FUNCTION "COOLANT" : VOID	// FC 50
TITLE = Coolant high pressure-KmDruckerhöhung
AUTHOR : A.Petz
VERSION : 0.6
VAR_INPUT
  iPnennV : INT ;	//Nenndruck des KmHochdruckventils bei 10V [Bar]
  iPMin : INT ;	//Min-Grenze für Anwahl Druckstufe [Bar]
  iPMax : INT ;	//Max-Grenze für Anwahl Druckstufe [Bar]
  iAfl : BYTE ;	//Meßwertauflösung (0:11+Vz,1:12+Vz,2:13+Vz,3-FF:15+Vz)
  iRmoDs : BOOL ;	//Rückmeldungen an LPlc ohne direkte KmDruckschalterabfrage
  iRmoFls : BOOL ;	//Rückmeldungen an LPlc ohne direkte KmDurchfluss-Schalterabfrage
  iFixedPressure : BOOL ;	//Anwahl für Druckerhöhungsstation mit fester Druckstufe IKZ (=TRUE)
END_VAR
VAR_TEMP
  iPlc : STRUCT 	//Signale von LeitPLC (aus DB111)
   machine_on : BOOL ;	//vonLPlc:Maschine bereit
   workroomdoor : BOOL ;	//vonLPlc:Arbeitsraumtüren geschlossen+verriegelt
   alarm_quit : BOOL ;	//vonLPlc:Störung, Alarm quittieren (Alarm Cancel)
   x : BOOL ;	//vonLPlc:
   coo_backflow : BOOL ;	//vonLPlc:Kühlmittelrückförderpumpe läuft
   pneumatic_pressure : BOOL ;	//vonLPlc:Pneumatik-(Luft-)druck vorhanden
   xa : BOOL ;	//vonLPlc:
   xb : BOOL ;	//vonLPlc:
   strobe_coo_pressure : BOOL ;	//vonLPlc:Strobe Druckumschaltung
   x_1 : BOOL ;	//vonLPlc:
   x_2 : BOOL ;	//vonLPlc:
   x_3 : BOOL ;	//vonLPlc:
   x_4 : BOOL ;	//vonLPlc:
   x_5 : BOOL ;	//vonLPlc:
   x_6 : BOOL ;	//vonLPlc:
   x_7 : BOOL ;	//vonLPlc:
   coolant1_m8 : BOOL ;	//vonLPlc:Anford. Kühmittel 1 (M8), Niederdruck
   coolant2_m7 : BOOL ;	//vonLPlc:Anford. Kühmittel 2 (M7), Hochdruck
   spraygun : BOOL ;	//vonLPlc:Anford. Spülpistole
   flush_lasercover : BOOL ;	//vonLPlc:Anford.Spülung Laservermessungsabdeckung
   flush_workpiece1 : BOOL ;	//vonLPlc:Anford.für Dach=Werkstückspülung
   flush_pallet_carrier : BOOL ;	//vonLPlc:Anford.Tischspülung bei PalWechsel
   flush_workroomdoor : BOOL ;	//vonLPlc:Anford.Arbeitsraumtür spülen
   flush_setupstation : BOOL ;	//vonLPlc:Anford.Rüstplatzspülung(Vorrichtung)
   x_16 : BOOL ;	//vonLPlc:
   x_17 : BOOL ;	//vonLPlc:
   x_18 : BOOL ;	//vonLPlc:
   x_19 : BOOL ;	//vonLPlc:
   x_20 : BOOL ;	//vonLPlc:
   x_21 : BOOL ;	//vonLPlc:
   x_22 : BOOL ;	//vonLPlc:
   x_23 : BOOL ;	//vonLPlc:
   PSoll : BYTE ;	//vonLPlc:Anwahl Druckstufe, BCD
   resBy : BYTE ;	//vonLPlc:Reserve Anwahl Druckstufe
  END_STRUCT ;
  oPlc : STRUCT 	//Signale an LeitPLC (DB112)
   ack_coolant1_m8 : BOOL ;	//anLPlc:Kühlmittel 1 (Niederdruck) ok
   ack_coolant2_m7 : BOOL ;	//anLPlc:Kühlmittel 2 (Hochdruck) ok
   message_flag : BOOL ;	//anLPlc:Warnung an Bediener, zB.Wasserstand
   no_emergency_stop : BOOL ;	//anLPlc:Fehler in Ksa, NotAus Masch.erforderlich
   no_spindle_feed_stop : BOOL ;	//anLPlc:Anford.SpiVs Halt durch Fehler in Ksa
   no_spindle_feed_stp_g0 : BOOL ;	//anLPlc:Anford.SpiVs Halt durch Fehler in Ksa bei nächst.G0
   no_diagnostic_alarm : BOOL ;	//anLPlc:Desina-Schalterüberwachung LOW-aktiv
   mode_auto : BOOL ;	//anLPlc:Kühlschmierstoffanlage in Betriebsart Automatik
   circuit_open_stop : BOOL ;	//anLPlc:Km Motorschutz gefallen, Masch.Halt
   circuit_open_msg : BOOL ;	//anLPlc:Km Motorschutz gefallen, Meldung
   x12 : BOOL ;	//anLPlc:Reserve Ksa max.Füllstand
   x13 : BOOL ;	//anLPlc:Reserve Ksa Warnung .min.Füllstand
   x14 : BOOL ;	//anLPlc:Reserve Ksa min.Füllstand, Masch.Halt
   x15 : BOOL ;	//anLPlc:Reserve Ksa Ende Papierbandfilter
   x16 : BOOL ;	//anLPlc:Reserve Ksa Warnung Ende Papierbandfilter
   x17 : BOOL ;	//anLPlc:Reserve
   PSoll : BYTE ;	//anLPlc:Rückmeldung Druckstufe, BCD
   resBy : BYTE ;	//anLPlc:Reserve Rückmeldung Druckstufe
  END_STRUCT ;
  s : STRUCT 	//statische da gerettete Lokaldaten
   PSoll : INT ;	//stat:letzter gespeicherter KmSolldruck
   PSollAlt : INT ;	//stat:letzter gespeich.KmSolldruck (alt, für Änderungserfassung)
   PSollAA : INT ;	//stat:letzter gespeich.KmSolldruck, berechnet für AA
   P20AA : INT ;	//stat:Solldruck 20Bar, berechnet für AA
   P40AA : INT ;	//stat:Solldruck 40Bar, berechnet für AA
   fk : ARRAY  [0 .. 15 ] OF //stat:Flankenhilfsmerker
   BOOL ;
   hvFEin : BOOL ;	//stat:KmHauptventil Fehler:Einschaltüberwachung
   hvFUnt : BOOL ;	//stat:KmHauptventil Fehler:Unterbrechungsüberwachung
   kmdFEin : BOOL ;	//stat:KmSystem=Niederdruck Fehler:Einschaltüberwachung
   kmdFUnt : BOOL ;	//stat:KmSystem=Niederdruck Fehler:Unterbrechungsüberwachung
   FlFEin : BOOL ;	//stat:KmDurchfluss Fehler:Einschaltüberwachung
   FlFUnt : BOOL ;	//stat:KmDurchfluss Fehler:Unterbrechungsüberwachung
   x_6 : BOOL ;	//stat:
   x_7 : BOOL ;	//stat:
   x_8 : BOOL ;	//stat:
   x_9 : BOOL ;	//stat:
   x_10 : BOOL ;	//stat:
   x_11 : BOOL ;	//stat:
   x_12 : BOOL ;	//stat:
   x_13 : BOOL ;	//stat:
   x_14 : BOOL ;	//stat:
   x_15 : BOOL ;	//stat:
  END_STRUCT ;
  svAR1 : DWORD ;	//Rettregister für AR1
  WertAA : INT ;	//Sollwert für Analogausgabe, ohne Meßwertauflösung
  LOp1 : BOOL ;	//lokaler Operationsmerker 1, Zwischenmerker
  LOp2 : BOOL ;	//lokaler Operationsmerker 2, Zwischenmerker
  LOp3 : BOOL ;	//lokaler Operationsmerker 3, Zwischenmerker
  fa : BOOL ;	//Freigabe Ausgänge
  no_coo_pressure : BOOL ;	//keine Km-Niederdruck Störung
  no_coo_flow : BOOL ;	//keine Km-Durchfluss Störung
  need_ventilate : BOOL ;	//Entlüftung wird benötigt
  ilp_ventilated : BOOL ;	//Anlage entlüftet
  shutdown_m7_opendoor : BOOL ;	//Abschaltung M7 über Öffnen der Arbeitsraumtüre
END_VAR
BEGIN
NETWORK
TITLE = Lokaldaten laden
      TAR1  #svAR1;
      LAR1  P##iPlc;
      L     DB111.DBD 0;
      T     LD [AR1,P#0.0];
      L     DB111.DBW 4;
      T     LW [AR1,P#4.0];
      LAR1  P##oPlc;
      L     DB112.DBW 0;
      T     LW [AR1,P#0.0];
      L     DB112.DBW 6;
      T     LW [AR1,P#2.0];
      LAR1  P##s;
      L     DB50.DBD 0;
      T     LD [AR1,P#0.0];
      L     DB50.DBD 4;
      T     LD [AR1,P#4.0];
      L     DB50.DBD 8;
      T     LD [AR1,P#8.0];
      L     DB50.DBW 12;
      T     LW [AR1,P#12.0];
      LAR1  #svAR1;
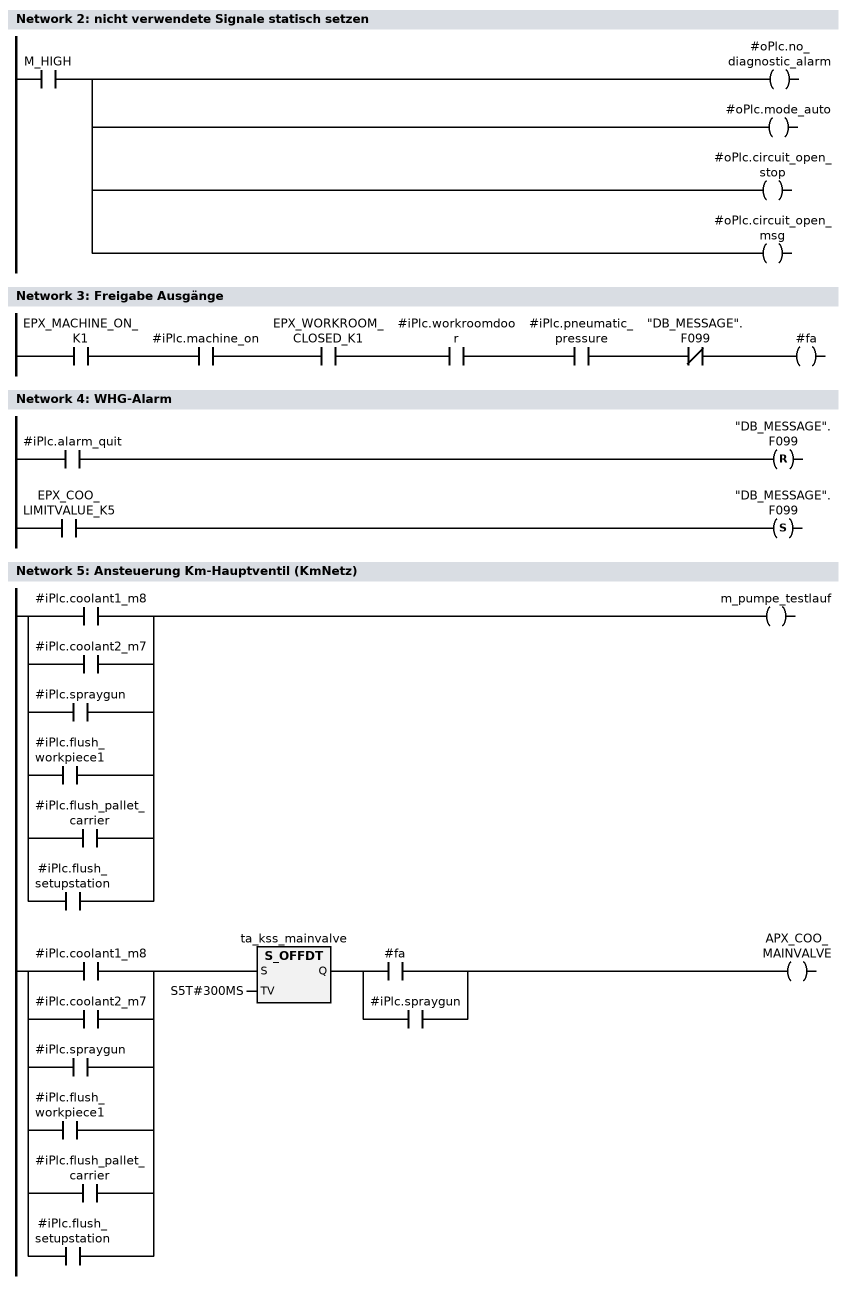
NETWORK
TITLE = nicht verwendete Signale statisch setzen 
      A     "M_HIGH";
      =     #oPlc.no_diagnostic_alarm;
      =     #oPlc.mode_auto;
      =     #oPlc.circuit_open_stop;
      =     #oPlc.circuit_open_msg;
NETWORK
TITLE = Freigabe Ausgänge
      A     "EPX_MACHINE_ON_K1";
      A     #iPlc.machine_on;
      A     "EPX_WORKROOM_CLOSED_K1";
      A     #iPlc.workroomdoor;
      A     #iPlc.pneumatic_pressure;
      AN    "DB_MESSAGE".F099;
      =     #fa;
NETWORK
TITLE = WHG-Alarm
      A     #iPlc.alarm_quit;
      R     "DB_MESSAGE".F099;
      A     "EPX_COO_LIMITVALUE_K5";
      S     "DB_MESSAGE".F099;
      NOP   0;
NETWORK
TITLE = Ansteuerung Km-Hauptventil (KmNetz)
//Bei Aktivierung der Sppritzpistole, wird nicht darauf geachtet ob die 
//Arbeitsraumtüren bzw. Rüstplatztüren geöffnet bzw. geschlossen sind, da dieses 
//PLC-seitig durchgeführt wird.
      O     #iPlc.coolant1_m8;
      O     #iPlc.coolant2_m7;
      O     #iPlc.spraygun;
      O     #iPlc.flush_workpiece1;
      O     #iPlc.flush_pallet_carrier;
      O     #iPlc.flush_setupstation;
      =     L 32.0;
      A(;
      A     L 32.0;
      L     S5T#300MS;
      SF    "ta_kss_mainvalve";
      NOP   0;
      NOP   0;
      NOP   0;
      A     "ta_kss_mainvalve";
      );
      A(;
      O     #fa;
      O     #iPlc.spraygun;
      );
      =     "APX_COO_MAINVALVE";
      A     L 32.0;
      BLD   102;
      =     "m_pumpe_testlauf";
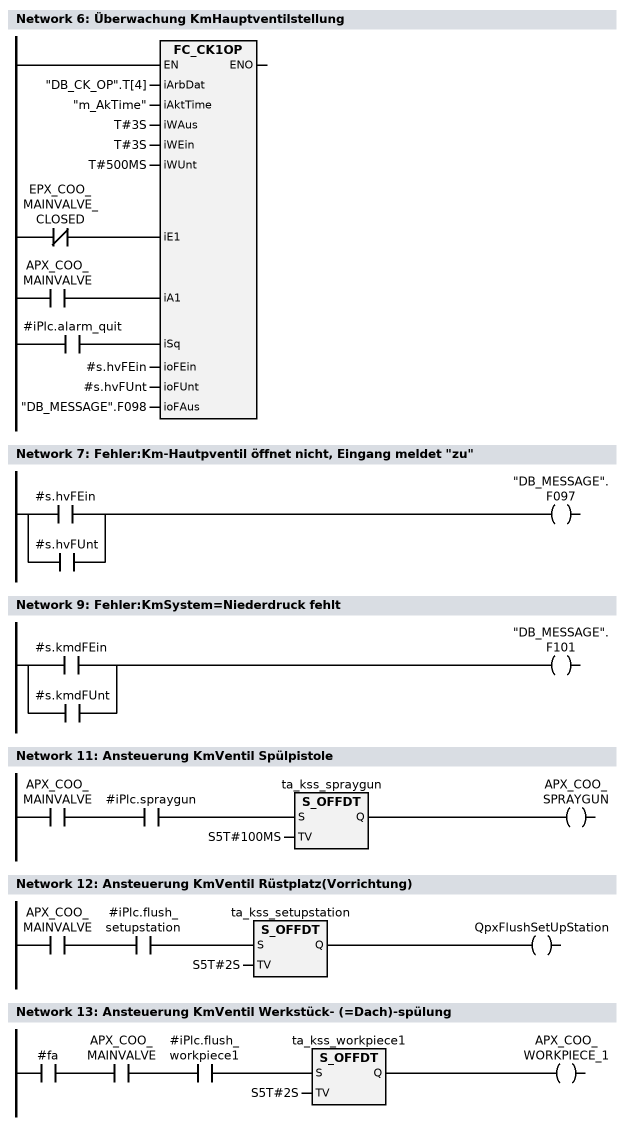
NETWORK
TITLE = Überwachung KmHauptventilstellung
//Koaxialventil
//Fabrikat: müller coax  Typ: 5-VMK32
//Das Ventil ist mit einem Endschalter ausgerüstet, welcher die 
//"geschlossen"-Position überwacht.
      AN    "EPX_COO_MAINVALVE_CLOSED";
      =     L 32.0;
      BLD   103;
      A     "APX_COO_MAINVALVE";
      =     L 32.1;
      BLD   103;
      A     #iPlc.alarm_quit;
      =     L 32.2;
      BLD   103;
      CALL  "FC_CK1OP" (
           iArbDat                  := "DB_CK_OP".T[4],
           iAktTime                 := "m_AkTime",
           iWAus                    := T#3S,
           iWEin                    := T#3S,
           iWUnt                    := T#500MS,
           iE1                      := L 32.0,
           iA1                      := L 32.1,
           iSq                      := L 32.2,
           ioFEin                   := #s.hvFEin,
           ioFUnt                   := #s.hvFUnt,
           ioFAus                   := "DB_MESSAGE".F098);
      NOP   0;
NETWORK
TITLE = Fehler:Km-Hautpventil öffnet nicht, Eingang meldet "zu"
//Koaxialventil
//Fabrikat: müller coax  Typ: 5-VMK32
//Das Ventil ist mit einem Endschalter ausgerüstet, welcher die 
//"geschlossen"-Position überwacht.
      O     #s.hvFEin;
      O     #s.hvFUnt;
      =     "DB_MESSAGE".F097;
NETWORK
TITLE = Überwachung KmSystem=Niederdruck
//Drucküberwachung wird zeitverzögert nach Entlüftung aktiviert, da die Anlage 
//Zeit zum Entlüften braucht.(Entlüftung nur bei geschlossener Arbeitsraumtüre)
      A     "EPX_COO_PRESSURE_P=MAX";
      A     "EPX_MACHINE_ON_K1";
      =     L 32.0;
      BLD   103;
      A     "APX_COO_MAINVALVE";
      =     L 32.1;
      BLD   103;
      A     #iPlc.alarm_quit;
      =     L 32.2;
      BLD   103;
      A(;
      A(;
      A     "ta_pressureless";
      L     S5T#1S;
      SD    "te_aktiv_monit_pressure";
      NOP   0;
      NOP   0;
      NOP   0;
      A     "te_aktiv_monit_pressure";
      );
      S     #ilp_ventilated;
      A     #need_ventilate;
      R     #ilp_ventilated;
      A     #ilp_ventilated;
      );
      JNB   _001;
      CALL  "FC_CK1OP" (
           iArbDat                  := "DB_CK_OP".T[5],
           iAktTime                 := "m_AkTime",
           iWAus                    := T#10S,
           iWEin                    := T#5S,
           iWUnt                    := T#2S,
           iE1                      := L 32.0,
           iA1                      := L 32.1,
           iSq                      := L 32.2,
           ioFEin                   := #s.kmdFEin,
           ioFUnt                   := #s.kmdFUnt,
           ioFAus                   := "DB_MESSAGE".F102);
_001: NOP   0;
NETWORK
TITLE = Fehler:KmSystem=Niederdruck fehlt
      O     #s.kmdFEin;
      O     #s.kmdFUnt;
      =     "DB_MESSAGE".F101;
NETWORK
TITLE = Aktivierung Kühlschmierstoffzufuhr_1 (externe - Spritzdüsen)
//Entlüftung der Anlage über M8 ist erst möglich wenn die Arbeitsraumtüre 
//geschlossen ist.
//Bei Abschaltung M7 über Türe öffnen wird ebenfalls ein Signal zur 
//erforderlichen 
//Entlüftung ausgegeben, da M7 Plc seitig nicht abfällt wenn Türe geöffnet wird.
      O(;
      A     #fa;
      A     "APX_COO_MAINVALVE";
      A     #iPlc.coolant1_m8;
      L     S5T#2S;
      SF    "ta_kss_km1";
      NOP   0;
      NOP   0;
      NOP   0;
      A     "ta_kss_km1";
      );
      O(;
      A(;
      A(;
      A(;
      A(;
      A     #iPlc.coolant2_m7;
      S     #shutdown_m7_opendoor;
      AN    #iPlc.workroomdoor;
      R     #shutdown_m7_opendoor;
      A     #shutdown_m7_opendoor;
      );
      FN    "m_fn_m7opendoor";
      O(;
      A(;
      O     #iPlc.coolant2_m7;
      O     #iPlc.flush_pallet_carrier;
      O     #iPlc.spraygun;
      );
      FN    "m_fn_m7S";
      );
      O(;
      A     "EPX_MACHINE_ON_K1";
      FP    "m_fp_masch_on";
      );
      );
      S     #need_ventilate;
      A     "ta_pressureless";
      R     #need_ventilate;
      A     #need_ventilate;
      );
      A     #iPlc.workroomdoor;
      L     S5T#2S;
      SF    "ta_pressureless";
      NOP   0;
      NOP   0;
      NOP   0;
      A     "ta_pressureless";
      );
      AN    "APX_COO_MAINVALVE";
      );
      =     "APX_COO_COOLANT1_(M8)";
NETWORK
TITLE = Ansteuerung KmVentil Spülpistole
      A     "APX_COO_MAINVALVE";
      A     #iPlc.spraygun;
      L     S5T#100MS;
      SF    "ta_kss_spraygun";
      NOP   0;
      NOP   0;
      NOP   0;
      A     "ta_kss_spraygun";
      =     "APX_COO_SPRAYGUN";
NETWORK
TITLE = Ansteuerung KmVentil Rüstplatz(Vorrichtung)
      A     "APX_COO_MAINVALVE";
      A     #iPlc.flush_setupstation;
      L     S5T#2S;
      SF    "ta_kss_setupstation";
      NOP   0;
      NOP   0;
      NOP   0;
      A     "ta_kss_setupstation";
      =     "QpxFlushSetUpStation";
NETWORK
TITLE = Ansteuerung KmVentil Werkstück- (=Dach)-spülung
      A     #fa;
      A     "APX_COO_MAINVALVE";
      A     #iPlc.flush_workpiece1;
      L     S5T#2S;
      SF    "ta_kss_workpiece1";
      NOP   0;
      NOP   0;
      NOP   0;
      A     "ta_kss_workpiece1";
      =     "APX_COO_WORKPIECE_1";
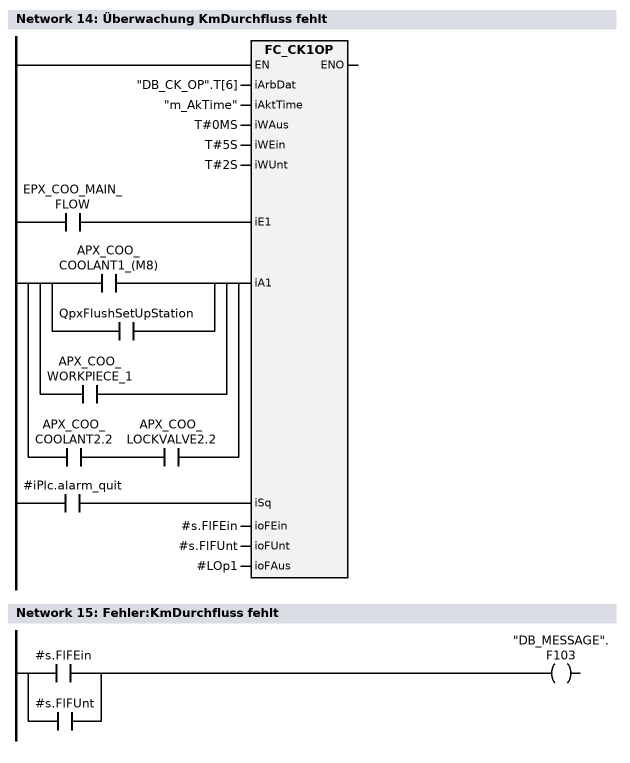
NETWORK
TITLE = Überwachung KmDurchfluss fehlt
      A     "EPX_COO_MAIN_FLOW";
      =     L 32.0;
      BLD   103;
      A(;
      O     "APX_COO_COOLANT1_(M8)";
      O     "QpxFlushSetUpStation";
      O     "APX_COO_WORKPIECE_1";
      O;
      A     "APX_COO_COOLANT2.2";
      A     "APX_COO_LOCKVALVE2.2";
      );
      =     L 32.1;
      BLD   103;
      A     #iPlc.alarm_quit;
      =     L 32.2;
      BLD   103;
      CALL  "FC_CK1OP" (
           iArbDat                  := "DB_CK_OP".T[6],
           iAktTime                 := "m_AkTime",
           iWAus                    := T#0MS,
           iWEin                    := T#5S,
           iWUnt                    := T#2S,
           iE1                      := L 32.0,
           iA1                      := L 32.1,
           iSq                      := L 32.2,
           ioFEin                   := #s.FlFEin,
           ioFUnt                   := #s.FlFUnt,
           ioFAus                   := #LOp1);
      NOP   0;
NETWORK
TITLE = Fehler:KmDurchfluss fehlt
      O     #s.FlFEin;
      O     #s.FlFUnt;
      =     "DB_MESSAGE".F103;
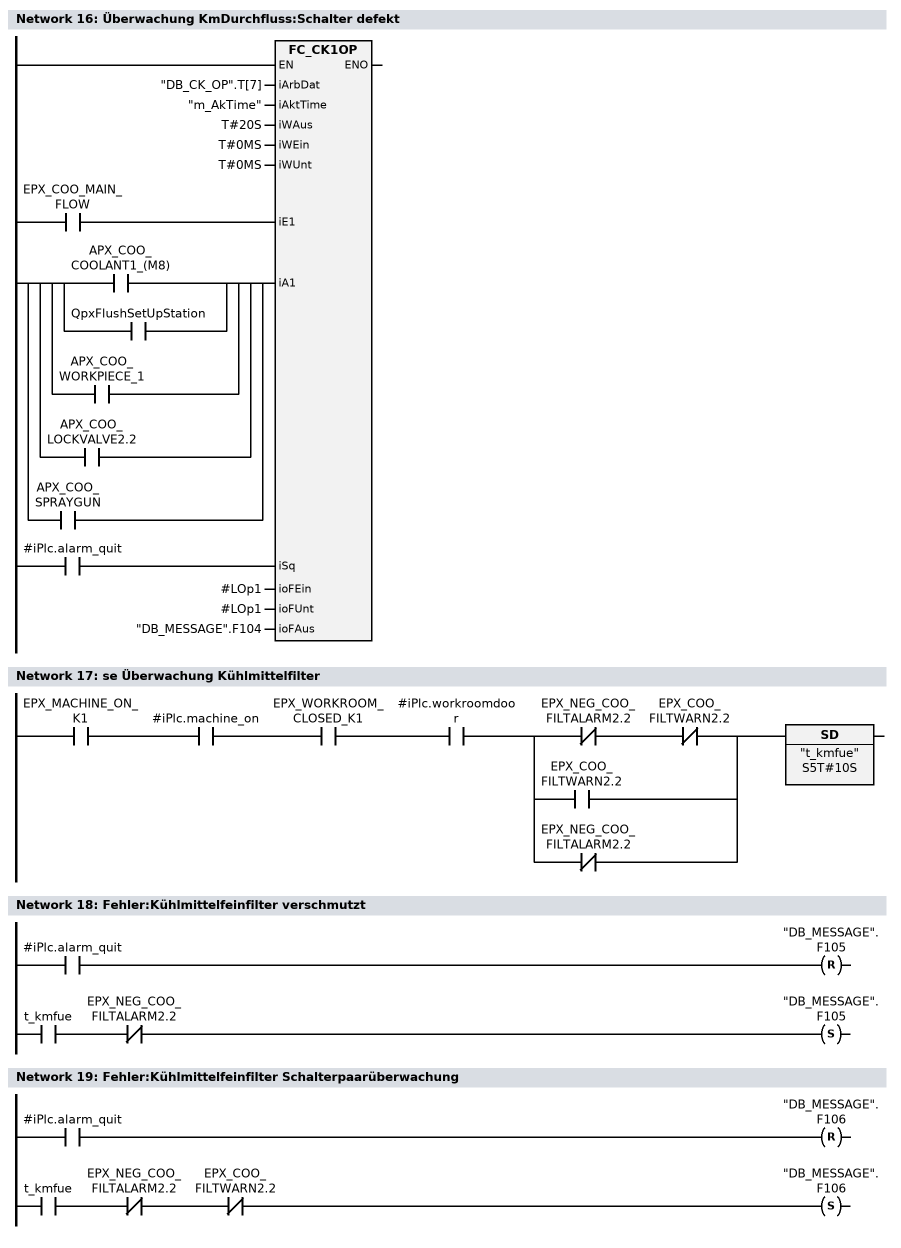
NETWORK
TITLE = Überwachung KmDurchfluss:Schalter defekt
      A     "EPX_COO_MAIN_FLOW";
      =     L 32.0;
      BLD   103;
      A(;
      O     "APX_COO_COOLANT1_(M8)";
      O     "QpxFlushSetUpStation";
      O     "APX_COO_WORKPIECE_1";
      O     "APX_COO_LOCKVALVE2.2";
      O     "APX_COO_SPRAYGUN";
      );
      =     L 32.1;
      BLD   103;
      A     #iPlc.alarm_quit;
      =     L 32.2;
      BLD   103;
      CALL  "FC_CK1OP" (
           iArbDat                  := "DB_CK_OP".T[7],
           iAktTime                 := "m_AkTime",
           iWAus                    := T#20S,
           iWEin                    := T#0MS,
           iWUnt                    := T#0MS,
           iE1                      := L 32.0,
           iA1                      := L 32.1,
           iSq                      := L 32.2,
           ioFEin                   := #LOp1,
           ioFUnt                   := #LOp1,
           ioFAus                   := "DB_MESSAGE".F104);
      NOP   0;
NETWORK
TITLE = se Überwachung Kühlmittelfilter
      A     "EPX_MACHINE_ON_K1";
      A     #iPlc.machine_on;
      A     "EPX_WORKROOM_CLOSED_K1";
      A     #iPlc.workroomdoor;
      A(;
      AN    "EPX_NEG_COO_FILTALARM2.2";
      AN    "EPX_COO_FILTWARN2.2";
      O     "EPX_COO_FILTWARN2.2";
      ON    "EPX_NEG_COO_FILTALARM2.2";
      );
      L     S5T#10S;
      SD    "t_kmfue";
NETWORK
TITLE = Fehler:Kühlmittelfeinfilter verschmutzt
      A     #iPlc.alarm_quit;
      R     "DB_MESSAGE".F105;
      A     "t_kmfue";
      AN    "EPX_NEG_COO_FILTALARM2.2";
      S     "DB_MESSAGE".F105;
      NOP   0;
NETWORK
TITLE = Fehler:Kühlmittelfeinfilter Schalterpaarüberwachung
      A     #iPlc.alarm_quit;
      R     "DB_MESSAGE".F106;
      A     "t_kmfue";
      AN    "EPX_NEG_COO_FILTALARM2.2";
      AN    "EPX_COO_FILTWARN2.2";
      S     "DB_MESSAGE".F106;
      NOP   0;
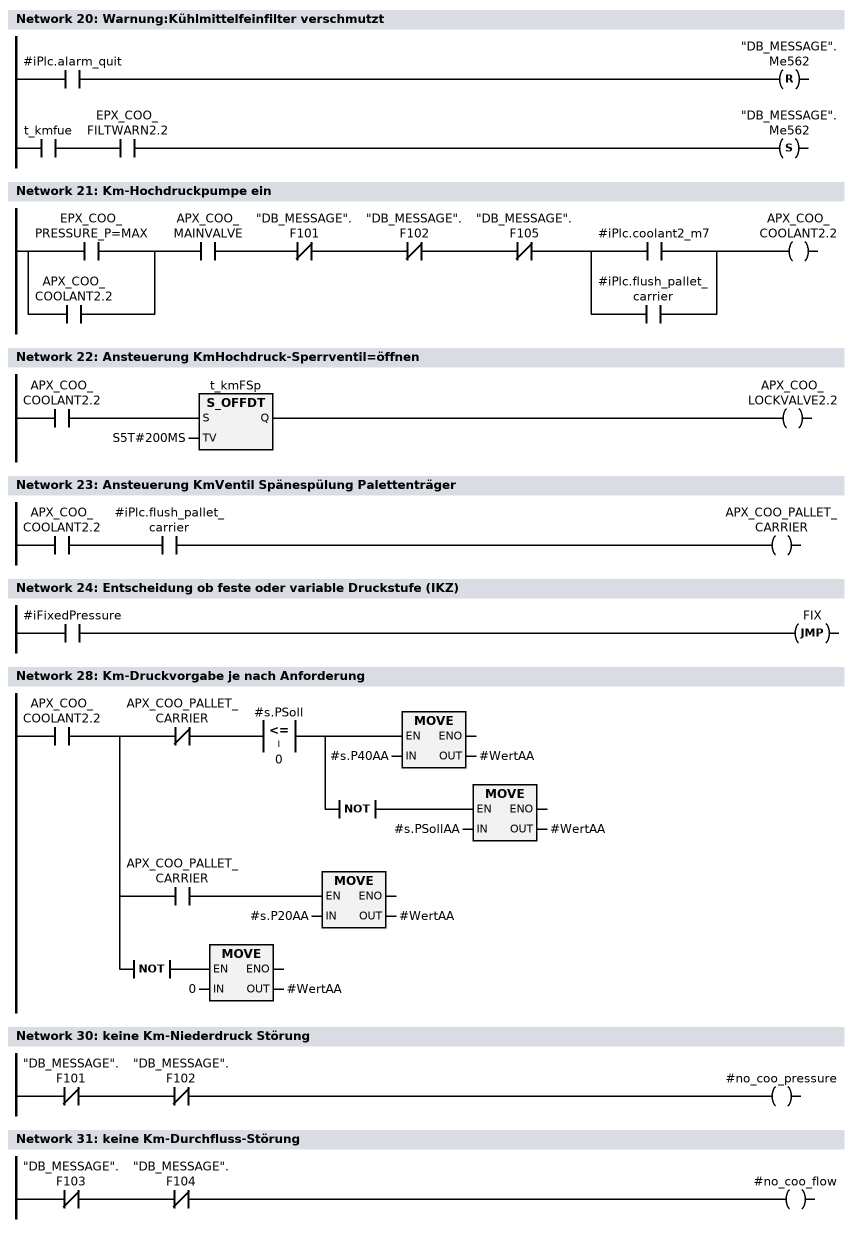
NETWORK
TITLE = Warnung:Kühlmittelfeinfilter verschmutzt
      A     #iPlc.alarm_quit;
      R     "DB_MESSAGE".Me562;
      A     "t_kmfue";
      A     "EPX_COO_FILTWARN2.2";
      S     "DB_MESSAGE".Me562;
      NOP   0;
NETWORK
TITLE = Km-Hochdruckpumpe ein
      A(;
      O     "EPX_COO_PRESSURE_P=MAX";
      O     "APX_COO_COOLANT2.2";
      );
      A     "APX_COO_MAINVALVE";
      AN    "DB_MESSAGE".F101;
      AN    "DB_MESSAGE".F102;
      AN    "DB_MESSAGE".F105;
      A(;
      O     #iPlc.coolant2_m7;
      O     #iPlc.flush_pallet_carrier;
      );
      =     "APX_COO_COOLANT2.2";
NETWORK
TITLE = Ansteuerung KmHochdruck-Sperrventil=öffnen
      A     "APX_COO_COOLANT2.2";
      L     S5T#200MS;
      SF    "t_kmFSp";
      NOP   0;
      NOP   0;
      NOP   0;
      A     "t_kmFSp";
      =     "APX_COO_LOCKVALVE2.2";
NETWORK
TITLE = Ansteuerung KmVentil Spänespülung Palettenträger
      A     "APX_COO_COOLANT2.2";
      A     #iPlc.flush_pallet_carrier;
      =     "APX_COO_PALLET_CARRIER";
NETWORK
TITLE = Entscheidung ob feste oder variable Druckstufe (IKZ)
      A     #iFixedPressure;
      JC    FIX;
NETWORK
TITLE = Km-Drucksollwertübernahme von LeitPlc (LPlc) übernehmen
      AN    #iPlc.strobe_coo_pressure;
      JC    e001;
//      L     #iPlc.PSoll
      L     DB111.DBW 4;
      BTI;
//---(1)--- Prüfung:Wert in zulässigem Bereich? --------
      L     #iPMin;
      <I;
      AN    #iFixedPressure;
      S     "DB_MESSAGE".Me563;
      JC    e001;
      TAK;
      L     #iPMax;
      >I;
      AN    #iFixedPressure;
      S     "DB_MESSAGE".Me563;
      JC    e001;
//---(1)------------------------------------------------
//---(2)--- Übernahme des Sollwertes und Rückmeldung an LPlc ---
      R     "DB_MESSAGE".Me563;
      TAK;
      T     #s.PSoll;
      ITB;
      T     #oPlc.PSoll;
//---(2)--------------------------------------------------------
e001: A     #iPlc.alarm_quit;
      R     "DB_MESSAGE".Me563;
NETWORK
TITLE = Wert berechnen für Analogausgabe bei Sollwertänderung
      L     #s.PSollAlt;
      L     #s.PSoll;
      ==I;
      JC    e002;
      T     #s.PSollAlt;
      DTR;
      L     #iPnennV;
      DTR;
      /R;
      L     2.764800e+04;
      *R;
      RND;
      T     #s.PSollAA;
e002: NOP   0;
NETWORK
TITLE = 20+40Bar Wert berechnen für AA bei Einschalten KmHochdruck
      A     "APX_COO_COOLANT2.2";
      FP    #s.fk[0];
      JCN   e003;
      L     20;	//Solldruck 20 Bar
      DTR;
      L     #iPnennV;
      DTR;
      /R;
      L     2.764800e+04;
      *R;
      RND;
      T     #s.P20AA;
      L     40;	//Solldruck 40 Bar
      DTR;
      L     #iPnennV;
      DTR;
      /R;
      L     2.764800e+04;
      *R;
      RND;
      T     #s.P40AA;
e003: NOP   0;
NETWORK
TITLE = Km-Druckvorgabe je nach Anforderung
      A     "APX_COO_COOLANT2.2";
      =     L 32.0;
      A     L 32.0;
      AN    "APX_COO_PALLET_CARRIER";
      A(;
      L     #s.PSoll;
      L     0;
      <=I;
      );
      =     L 32.1;
      A     L 32.1;
      JNB   _002;
      L     #s.P40AA;
      T     #WertAA;
_002: NOP   0;
      A     L 32.1;
      NOT;
      JNB   _003;
      L     #s.PSollAA;
      T     #WertAA;
_003: NOP   0;
      A     L 32.0;
      A     "APX_COO_PALLET_CARRIER";
      JNB   _010;
      L     #s.P20AA;
      T     #WertAA;
_010: NOP   0;
      A     L 32.0;
      NOT;
      JNB   _011;
      L     0;
      T     #WertAA;
_011: NOP   0;
NETWORK
TITLE = Sollwert an Meßwerauflösung der Analogausgabe (AA) anpassen
      L     #iAfl;
      JL    lstx;
      JU    sr00;
      JU    sr01;
      JU    sr02;
      JU    sr03;
lstx: JU    maxs;
sr00: L     W#16#FFF0;	//Maske bei 11Bit+Vz
      JU    w001;
sr01: L     W#16#FFF8;	//Maske bei 12Bit+Vz
      JU    w001;
sr02: L     W#16#FFFC;	//Maske bei 13Bit+Vz
      JU    w001;
sr03: L     W#16#FFFF;	//Maske bei 15Bit+Vz
      JU    w001;
maxs: L     W#16#FFFF;	//Werte >3 werden als 15Bit+Vz behandelt
w001: L     #WertAA;
      AW;
      T     "APW_COO_PRESS_VALUE2.2";
NETWORK
TITLE = keine Km-Niederdruck Störung
FIX:  AN    "DB_MESSAGE".F101;
      AN    "DB_MESSAGE".F102;
      =     #no_coo_pressure;
NETWORK
TITLE = keine Km-Durchfluss-Störung
      AN    "DB_MESSAGE".F103;
      AN    "DB_MESSAGE".F104;
      =     #no_coo_flow;
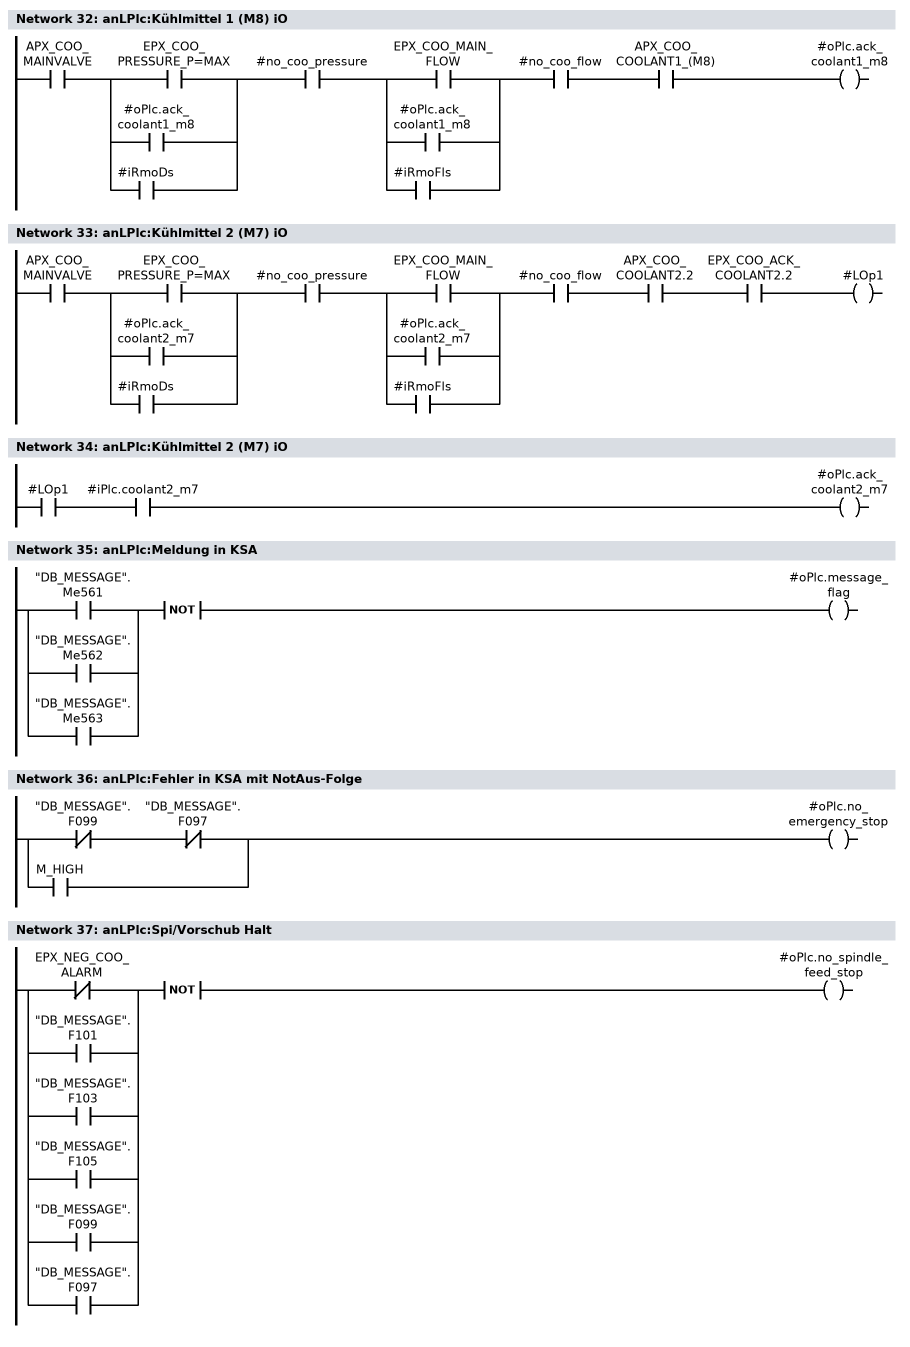
NETWORK
TITLE = anLPlc:Kühlmittel 1 (M8) iO
      A     "APX_COO_MAINVALVE";
      A(;
      O     "EPX_COO_PRESSURE_P=MAX";
      O     #oPlc.ack_coolant1_m8;
      O     #iRmoDs;
      );
      A     #no_coo_pressure;
      A(;
      O     "EPX_COO_MAIN_FLOW";
      O     #oPlc.ack_coolant1_m8;
      O     #iRmoFls;
      );
      A     #no_coo_flow;
      A     "APX_COO_COOLANT1_(M8)";
      =     #oPlc.ack_coolant1_m8;
NETWORK
TITLE = anLPlc:Kühlmittel 2 (M7) iO
      A     "APX_COO_MAINVALVE";
      A(;
      O     "EPX_COO_PRESSURE_P=MAX";
      O     #oPlc.ack_coolant2_m7;
      O     #iRmoDs;
      );
      A     #no_coo_pressure;
      A(;
      O     "EPX_COO_MAIN_FLOW";
      O     #oPlc.ack_coolant2_m7;
      O     #iRmoFls;
      );
      A     #no_coo_flow;
      A     "APX_COO_COOLANT2.2";
      A     "EPX_COO_ACK_COOLANT2.2";
      =     #LOp1;
NETWORK
TITLE = anLPlc:Kühlmittel 2 (M7) iO
      A     #LOp1;
      A     #iPlc.coolant2_m7;
      =     #oPlc.ack_coolant2_m7;
NETWORK
TITLE = anLPlc:Meldung in KSA
      A(;
      O     "DB_MESSAGE".Me561;
      O     "DB_MESSAGE".Me562;
      O     "DB_MESSAGE".Me563;
      );
      NOT;
      =     #oPlc.message_flag;
NETWORK
TITLE = anLPlc:Fehler in KSA mit NotAus-Folge
      AN    "DB_MESSAGE".F099;
      AN    "DB_MESSAGE".F097;
      O     "M_HIGH";
      =     #oPlc.no_emergency_stop;
NETWORK
TITLE = anLPlc:Spi/Vorschub Halt
      A(;
      ON    "EPX_NEG_COO_ALARM";
      O     "DB_MESSAGE".F101;
      O     "DB_MESSAGE".F103;
      O     "DB_MESSAGE".F105;
      O     "DB_MESSAGE".F099;
      O     "DB_MESSAGE".F097;
      );
      NOT;
      =     #oPlc.no_spindle_feed_stop;
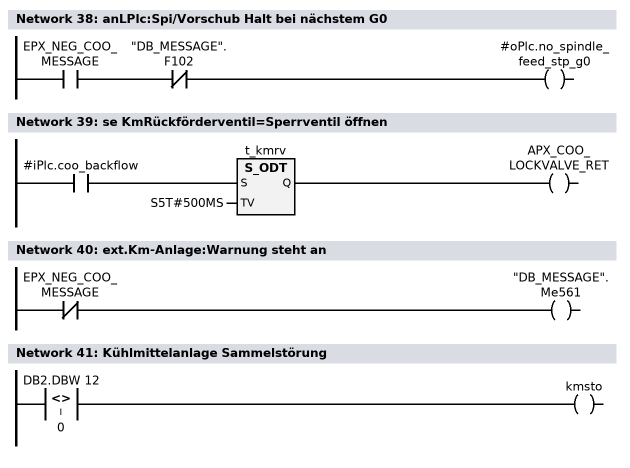
NETWORK
TITLE = anLPlc:Spi/Vorschub Halt bei nächstem G0
      A     "EPX_NEG_COO_MESSAGE";
      AN    "DB_MESSAGE".F102;
      =     #oPlc.no_spindle_feed_stp_g0;
NETWORK
TITLE = se KmRückförderventil=Sperrventil öffnen
      A     #iPlc.coo_backflow;
      L     S5T#500MS;
      SD    "t_kmrv";
      NOP   0;
      NOP   0;
      NOP   0;
      A     "t_kmrv";
      =     "APX_COO_LOCKVALVE_RET";
NETWORK
TITLE = ext.Km-Anlage:Warnung steht an
      AN    "EPX_NEG_COO_MESSAGE";
      =     "DB_MESSAGE".Me561;
NETWORK
TITLE = Kühlmittelanlage Sammelstörung
      L     DB2.DBW 12;
      L     0;
      <>I;
      =     "kmsto";
NETWORK
TITLE = Lokaldaten retten
      TAR1  #svAR1;
      LAR1  P##oPlc;
      L     LW [AR1,P#0.0];
      T     DB112.DBW 0;
      L     LW [AR1,P#2.0];
      T     DB112.DBW 6;
      LAR1  P##s;
      L     LD [AR1,P#0.0];
      T     DB50.DBD 0;
      L     LD [AR1,P#4.0];
      T     DB50.DBD 4;
      L     LD [AR1,P#8.0];
      T     DB50.DBD 8;
      L     LW [AR1,P#12.0];
      T     DB50.DBW 12;
      LAR1  #svAR1;
END_FUNCTION

FUNCTION "FUNCTIONS" : VOID	// FC 90
TITLE = Funktionen für Sonderanwendungen
//Funktion_1 ... Auswerten von Maschinenparametern (int_id =1)
//
AUTHOR : APetz
VERSION : 0.1
VAR_INPUT
  IN_INT_IDENTIFICATION : INT ;	//Auswahl der Funktion
  IN_WRD_PARAMETER : WORD ;	//z.B. Maschinenparameter
  IN_INT_DEKADE : INT ;	//Auswahl der Dekade <Dekade_4><Dekade_3><Dekade_2><Dekade_1>
  IN_INT_WERT : INT ;	//Angabe des Wertes, mit welchem verglichen werden soll
  IN_BIT_BYTE : BOOL ;	//Auswahl des Rückgabewertes für HIGH-Byte=0 oder des LOW-Bytes=1
END_VAR
VAR_OUTPUT
  OUT_BIT_PRUEF : BOOL ;	//Rückgabewert für Wertvergleich in Dekade
  OUT_BYT_WERT : BYTE ;	//Wert von Dekade bzw. HIGH- oder LOW-Byte des Maschinenparameters
END_VAR
BEGIN
NETWORK
TITLE = Auswerten von Dekaden eines Wortes (int_id = 1)
//Definition der Dekaden eines Wortes (4/3/2/1)
//Mittels dieser Funktion kann überprüft werden, ob eine beliebiger "Wert" (0 .. 
//9) <IN_INT_WERT> in einer beliebigen "Dekade" (1 ... 4) <IN_INT_DEKADE> im 
//Maschinenparameter "MP" <IN_WRD_PARAMETER> gesetzt wurde. Als Ergebnis wird der 
//Wert TRUE oder FALSE im <OUT_BIT_PRÜFUNG> zurückgegeben.
//Entspricht der übergebene Parameter in Dekade nicht 1 ... 4 wird FALSE 
//zurückgegeben.
//EN-Eingang gesetzt (bei KOP/FUP)?
      A     BR;
      JCN   END;
      L     #IN_INT_IDENTIFICATION;
      L     1;
      ==I;
      JCN   N_2;
      L     #IN_INT_DEKADE;	//lade Wert in Akku1-L-L
      JL    N_1Z;	//Akku1-L-L > 4
      JU    N_1Z;	//Akku1-L-L = 0 
      JU    N_1A;	//Akku1-L-L = 1
      JU    N_1B;	//Akku1-L-L = 2
      JU    N_1C;	//Akku1-L-L = 3
      JU    N_1D;	//Akku1-L-L = 4
//... ungültige Werte
N_1Z: SET;
      L     0;
      T     #OUT_BYT_WERT;
      R     #OUT_BIT_PRUEF;
      JU    N_E1;
//... Dekade 1
N_1A: L     #IN_WRD_PARAMETER;
      ITD;
      DTB;
      SLD   28;
      SRD   28;
      BTD;
      L     #IN_INT_WERT;
      ==I;
      =     #OUT_BIT_PRUEF;
      JU    N_E1;
//... Dekade 2
N_1B: L     #IN_WRD_PARAMETER;
      ITD;
      DTB;
      SLD   24;
      SRD   28;
      BTD;
      L     #IN_INT_WERT;
      ==I;
      =     #OUT_BIT_PRUEF;
      JU    N_E1;
//... Dekade 3
N_1C: L     #IN_WRD_PARAMETER;
      ITD;
      DTB;
      SLD   20;
      SRD   28;
      BTD;
      L     #IN_INT_WERT;
      ==I;
      =     #OUT_BIT_PRUEF;
      JU    N_E1;
//... Dekade 4
N_1D: L     #IN_WRD_PARAMETER;
      ITD;
      DTB;
      SLD   16;
      SRD   28;
      BTD;
      L     #IN_INT_WERT;
      ==I;
      =     #OUT_BIT_PRUEF;
      JU    N_E1;
N_E1: NOP   0;
//Funktion wurde korrekt ausgeführt
//setzt ENO auf High
      SET;
      SAVE;
      BE;
NETWORK
TITLE =
//Beim Aufruf dieser Funktion wird der Wert aus einer beliebigen "Dekade" (1 ... 
//4) <IN_INT_DEKADE> im Maschinenparameter "MP" <IN_WRD_PARAMETER> ausgelesen und 
//des-sen Wert in <OUT_BYT_WERT> zurückgegeben.
N_2:  L     #IN_INT_IDENTIFICATION;
      L     2;
      ==I;
      JCN   N_3;
      L     #IN_INT_DEKADE;	//lade Wert in Akku1-L-L
      JL    N_2Z;	//Akku1-L-L > 4
      JU    N_2Z;	//Akku1-L-L = 0 
      JU    N_2A;	//Akku1-L-L = 1
      JU    N_2B;	//Akku1-L-L = 2
      JU    N_2C;	//Akku1-L-L = 3
      JU    N_2D;	//Akku1-L-L = 4
//... ungültige Werte
N_2Z: SET;
      L     0;
      T     #OUT_BYT_WERT;
      R     #OUT_BIT_PRUEF;
      JU    N_E2;
//... Dekade 1
N_2A: L     #IN_WRD_PARAMETER;
      ITD;
      DTB;
      SLD   28;
      SRD   28;
      BTD;
      T     #OUT_BYT_WERT;
      JU    N_E2;
//... Dekade 2
N_2B: L     #IN_WRD_PARAMETER;
      ITD;
      DTB;
      SLD   24;
      SRD   28;
      BTD;
      T     #OUT_BYT_WERT;
      JU    N_E2;
//... Dekade 3
N_2C: L     #IN_WRD_PARAMETER;
      ITD;
      DTB;
      SLD   20;
      SRD   28;
      BTD;
      T     #OUT_BYT_WERT;
      JU    N_E2;
//... Dekade 4
N_2D: L     #IN_WRD_PARAMETER;
      ITD;
      DTB;
      SLD   16;
      SRD   28;
      BTD;
      T     #OUT_BYT_WERT;
      JU    N_E2;
N_E2: NOP   0;
//Funktion wurde korrekt ausgeführt
//setzt ENO auf High
      SET;
      SAVE;
      BE;
NETWORK
TITLE =
//Die Funktion ermittelt den Wert des <IN_BIT_BYTE> HIGH-Bytes oder des LOW-Bytes 
//im Maschinenparameter "MP" <IN_WRD_PARAMETER> und gibt diesen in <OUT_BYT_WERT> 
//zurück
N_3:  L     #IN_INT_IDENTIFICATION;
      L     3;
      ==I;
      JCN   END;	//Wenn VKE = 0 -->  springt an das Sprungziel.
      A     #IN_BIT_BYTE;	//Selektion HIGH-Byte (IN_BIT_BYTE = 0)
      JC    N_31;	//Wenn VKE = 1 -->  springt an das Sprungziel.   
      L     #IN_WRD_PARAMETER;	//lade Wert in Akku1-L-L
      ITD;	//lädt den Inhalt des in AKKU 1
      DTB;
      SLD   16;
      SRD   24;
      BTD;
      T     #OUT_BYT_WERT;
      JU    N_E3;
N_31: L     #IN_WRD_PARAMETER;	//lade Wert in Akku1-L-L
      ITD;	//lädt den Inhalt des in AKKU 1
      DTB;
      SLD   24;
      SRD   24;
      BTD;
      T     #OUT_BYT_WERT;
N_E3: NOP   0;
//Funktion wurde korrekt ausgeführt
//setzt ENO auf High
      SET;
      SAVE;
      BE;
END:  NOP   0;
//Enable beim Aufruf = 0 --> ENO-Ausgang auch auf 0 setzen
      CLR;
      SAVE;
END_FUNCTION

FUNCTION "CHANGE_BYTE" : VOID	// FC 91
//FUNKTION 1:
//
AUTHOR : A.Petz
VERSION : 0.1
VAR_INPUT
  I_ID : INT ;	//Identifikation der Funktion (Integer)
  W_MP : WORD ;	//Wert des Maschinenparameters
END_VAR
VAR_OUTPUT
  W_CHANGE_MP : WORD ;	//Wert des Maschinenparameters (angepasst an Reihenfolge der Bytes)
END_VAR
BEGIN
NETWORK
TITLE =
//Kehrt die Reihenfolge der Bytes in AKKU1-L
//Das Ergebnis wird in AKKU1-L gespeichert
//EN-Eingang gesetzt (bei KOP/FUP)?
//      U     BIE
//      SPBN  END1
      L     #I_ID;
      L     1;
      ==I;
      JCN   N_E1;
      L     #W_MP;
      CAW;
      T     #W_CHANGE_MP;
N_E1: NOP   0;
//Funktion wurde korrekt ausgeführt
//setzt ENO auf High
      SET;
      SAVE;
END_FUNCTION

FUNCTION "SIGNAL" : VOID	// FC 92
TITLE = ALLGEMEINE SIGNALVERKNÜPFUNGEN
//Funktionen zum Bilden von diversen Signalverknüpfungen, die für 
//unterschiedliche Anwendungen verwendet werden können (z.B. 
//Betriebsdatenerfassung, Signalleuchte, ...)
AUTHOR : A.Petz
VERSION : 0.1
VAR_INPUT
  IN_INT_IDENTIFICATION : INT ;	//Funktionskennung der Signalverküpfung
END_VAR
VAR_OUTPUT
  OUT_BIT_SIGNAL : BOOL ;	//Ergebnis der Signalverknüpfung
END_VAR
VAR_TEMP
  TMP_INT_IDENTIFICATION : INT ;	//Identifiaktionsnummer der Funktion
  TMP_BIT_ENABLE : BOOL ;	//Bausteinfreigabe - Sammelstörung
END_VAR
BEGIN
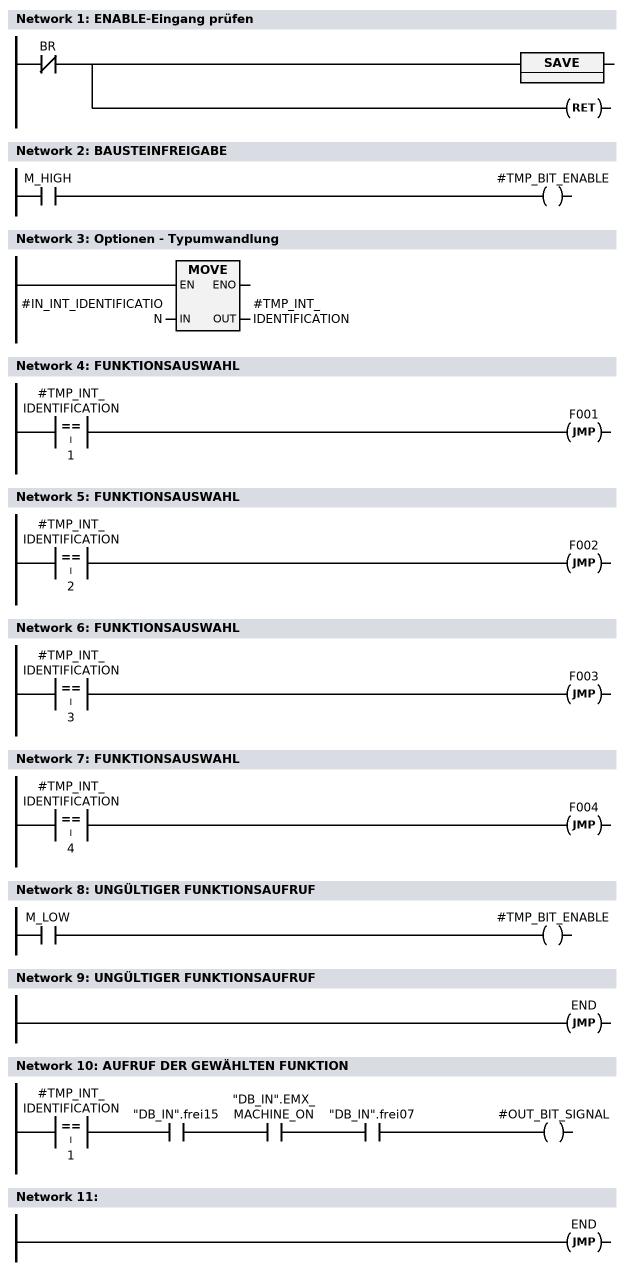
NETWORK
TITLE = ENABLE-Eingang prüfen
//Auswerten des BIE-Statusbit. Dieses entspricht dem EN (ENABLE)-Einganges bei 
//KOP/FUP. Wenn EN=FALSE dann verlasse Baustein.
      AN    BR;
      SAVE;
      BEC;
NETWORK
TITLE = BAUSTEINFREIGABE
//Fehlerauswertung Baustein intern:
//Bausteinfreigabe wird gesetzt
      A     "M_HIGH";
      =     #TMP_BIT_ENABLE;
NETWORK
TITLE = Optionen - Typumwandlung
//Konvertierung des "Identifikationsbytes" nach Integer
      L     #IN_INT_IDENTIFICATION;
      T     #TMP_INT_IDENTIFICATION;
      NOP   0;
NETWORK
TITLE = FUNKTIONSAUSWAHL
//Funktion mit Identifikation = 1 aufrufen
//Spindel läuft und mindestens eine Achse in Bewegung
//... wird bei "Not-Aus" zurückgesetzt.
      L     #TMP_INT_IDENTIFICATION;
      L     1;
      ==I;
      JC    F001;
NETWORK
TITLE = FUNKTIONSAUSWAHL
//Funktion mit Identifikation = 2 aufrufen
//Betriebsart MDA (Teach-In), SINGLE oder Betriebsart AUTOMATIK angewählt und 
//Programm läuft.
//... wird bei "Not-Aus" zurückgesetzt.
      L     #TMP_INT_IDENTIFICATION;
      L     2;
      ==I;
      JC    F002;
NETWORK
TITLE = FUNKTIONSAUSWAHL
//Funktion mit Identifikation = 3 aufrufen
//Maschine Ein und Betriebsart MANUAL angewählt.
      L     #TMP_INT_IDENTIFICATION;
      L     3;
      ==I;
      JC    F003;
NETWORK
TITLE = FUNKTIONSAUSWAHL
//Funktion mit Identifikation = 4 aufrufen
//Maschinenstörung (Fehlermeldung) oder Programm Ende oder Not-Aus
      L     #TMP_INT_IDENTIFICATION;
      L     4;
      ==I;
      JC    F004;
NETWORK
TITLE = UNGÜLTIGER FUNKTIONSAUFRUF
//Wenn keine gültige Identifikationsnummer übergeben wurde, wird das 
//Bausteinfreigabe (Sammelstörmeldung-Baustein) zurückgesetzt.
      A     "M_LOW";
      =     #TMP_BIT_ENABLE;
NETWORK
TITLE = UNGÜLTIGER FUNKTIONSAUFRUF
//Wenn keine gültige Identifikationsnummer übergeben wurde, wird an das 
//Programm-Ende gesprungen.
      JU    END;
NETWORK
TITLE = AUFRUF DER GEWÄHLTEN FUNKTION
//IDENTIFICATION = 1
//Spindel läuft und mindestens eine Achse in Bewegung
//... wird bei "Not-Aus" zurückgesetzt.
F001: A(;
      L     #TMP_INT_IDENTIFICATION;
      L     1;
      ==I;
      );
      A     "DB_IN".frei15;
      A     "DB_IN".EMX_MACHINE_ON;
      A     "DB_IN".frei07;
      =     #OUT_BIT_SIGNAL;
NETWORK
TITLE =
      JU    END;	//      BEA   
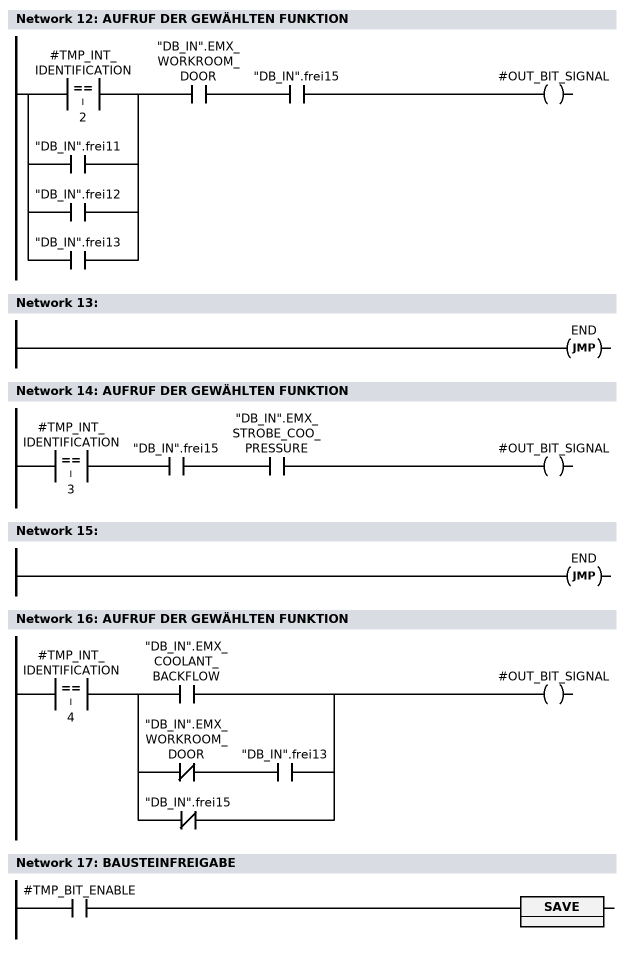
NETWORK
TITLE = AUFRUF DER GEWÄHLTEN FUNKTION
//IDENTIFICATION = 2
//Betriebsart MDA (Teach-In), SINGLE oder Betriebsart AUTOMATIK angewählt und 
//Programm läuft.
//... wird bei "Not-Aus" zurückgesetzt.
F002: A(;
      O(;
      L     #TMP_INT_IDENTIFICATION;
      L     2;
      ==I;
      );
      O     "DB_IN".frei11;
      O     "DB_IN".frei12;
      O     "DB_IN".frei13;
      );
      A     "DB_IN".EMX_WORKROOM_DOOR;
      A     "DB_IN".frei15;
      =     #OUT_BIT_SIGNAL;
NETWORK
TITLE =
      JU    END;	//      BEA   
NETWORK
TITLE = AUFRUF DER GEWÄHLTEN FUNKTION
//IDENTIFICATION = 3
//Maschine Ein und Betriebsart MANUAL angewählt.
F003: A(;
      L     #TMP_INT_IDENTIFICATION;
      L     3;
      ==I;
      );
      A     "DB_IN".frei15;
      A     "DB_IN".EMX_STROBE_COO_PRESSURE;
      =     #OUT_BIT_SIGNAL;
NETWORK
TITLE =
      JU    END;	//      BEA   
NETWORK
TITLE = AUFRUF DER GEWÄHLTEN FUNKTION
//IDENTIFICATION = 4
//Maschinenstörung (Fehlermeldung) oder Programm Ende (in Betriebsart 
//"Automatik") oder Not-Aus
F004: A(;
      L     #TMP_INT_IDENTIFICATION;
      L     4;
      ==I;
      );
      A(;
      O     "DB_IN".EMX_COOLANT_BACKFLOW;
      O;
      AN    "DB_IN".EMX_WORKROOM_DOOR;
      A     "DB_IN".frei13;
      ON    "DB_IN".frei15;
      );
      =     #OUT_BIT_SIGNAL;
NETWORK
TITLE = BAUSTEINFREIGABE
//Statusbit BIE=ENO setzen, wenn Funktion ohne Fehler durchlaufen wurde.
END:  A     #TMP_BIT_ENABLE;
      SAVE;
END_FUNCTION

FUNCTION "FC_CK2OP" : VOID	// FC 101
TITLE = Überwachung von 2 Aus-/Eingängen
//________________________________________________________________________________
//$Revision: x.y $
//$Date: 2005/04/26 0:0:0CET $
//$Author: slh $
//$ProjectRevision: Last Checkpoint: m.n $
//
//-------------------------------------------------------------------------------
//*ALL RIGHTS RESERVED
//*Softwareentwicklung
//erstellt: 09.05.2005; Helmut Scheuenstuhl (slh); Scheuenstuhl PAC / V0.1
//Änderung: Datum / Abteilung / Name / Version x.y
//Änderung: 
//        :
//-------------------------------------------------------------------------------
//Beschreibung
//Der Fc dient zur Überwachung von 2 Stellgliedern (Ventile o.ä.)
//Pro Aufruf werden 14 Byte Arbeitsdaten benötigt, deren Adresse über 
//iArbDat(Any) angegeben wird.
//WICHTIGE VORAUSSETZUNG:
//Der Fc arbeitet mit der Plc-Zeit, die mit SFC64 Time_tck ausgelesen und am
//"iAktTime" angeboten werden muß.
AUTHOR : SPAC_slh
FAMILY : Diagnose
NAME : CK2OP
VERSION : 0.1
VAR_INPUT
  iArbDat : ANY ;	//Rettadresse der 14Byte Arbeitsdaten des Fc
  iAktTime : TIME ;	//ausgeleseneSysZeitVonTime_tck SFC64
  iWPaar : TIME ;	//Verzögerung Paarüberwachung, T#0MS= Abwahl
  iWLz : TIME ;	//Verzögerung Laufzeitüberwachung, T#0MS= Abwahl
  iWEndl : TIME ;	//Verzögerung Endlagenüberwachung, T#0MS= Abwahl
  iE1 : BOOL ;	//Schalter, wird durch iA1 angefahren
  iA1 : BOOL ;	//zu überwachender Ausgang 1
  iE2 : BOOL ;	//Schalter, wird durch iA2 angefahren
  iA2 : BOOL ;	//zu überwachender Ausgang 2
  iDL : BOOL ;	//gespeicherte Endstlg.mit Befehl 0 abschalten
  iSq : BOOL ;	//Störung quittieren
  iNoPaar : BOOL ;	//Paarüberwachung abschalten
  iNoLz : BOOL ;	//Laufzeitüberwachung abschalten
  iNoEnd : BOOL ;	//Endlagenüberwachung abschalten
END_VAR
VAR_IN_OUT
  ioFLz1 : BOOL ;	//Laufzeitfehler bei Stlg.1 anfahren
  ioFLz2 : BOOL ;	//Laufzeitfehler bei Stlg.2 anfahren
  ioFEnd1 : BOOL ;	//Fehler:Endlage 1 wurde verlassen
  ioFEnd2 : BOOL ;	//Fehler:Endlage 2 wurde verlassen
  ioFPaar : BOOL ;	//Fehler Paarüberwachung
END_VAR
VAR_TEMP
  AdrArDat : ANY ;	//Übergabeparameter für Adresse der Arbeitsdaten
  svAr1 : DWORD ;
  svAr2 : DWORD ;
  s : UDT 1010;	//stat, da gerettet
  RetVal : INT ;
  Lop1 : BOOL ;
  seEingang : BOOL ;	//SwTimer se Eingang
  seFpEing : BOOL ;	//SwTimer se Eingang pos.Flanke
  seAbgel : BOOL ;	//SwTimer se abgelaufen
  seAusgang : BOOL ;	//SwTimer se Ausgang
  fpiA1 : BOOL ;
  fpiA2 : BOOL ;
  fpSq : BOOL ;	//Flanke Störung quittieren
END_VAR
BEGIN
NETWORK
TITLE = Übergabezeiger für BLKMOV aus iArbDat übernehmen
      TAR1  #svAr1;
      TAR2  #svAr2;
      L     P##iArbDat;
      LAR1;
      LAR2  P##AdrArDat;
      L     W [AR1,P#0.0];
      T     LW [AR2,P#0.0];
      L     D [AR1,P#2.0];
      T     LD [AR2,P#2.0];
      L     D [AR1,P#6.0];
      T     LD [AR2,P#6.0];
      LAR1  #svAr1;
      LAR2  #svAr2;
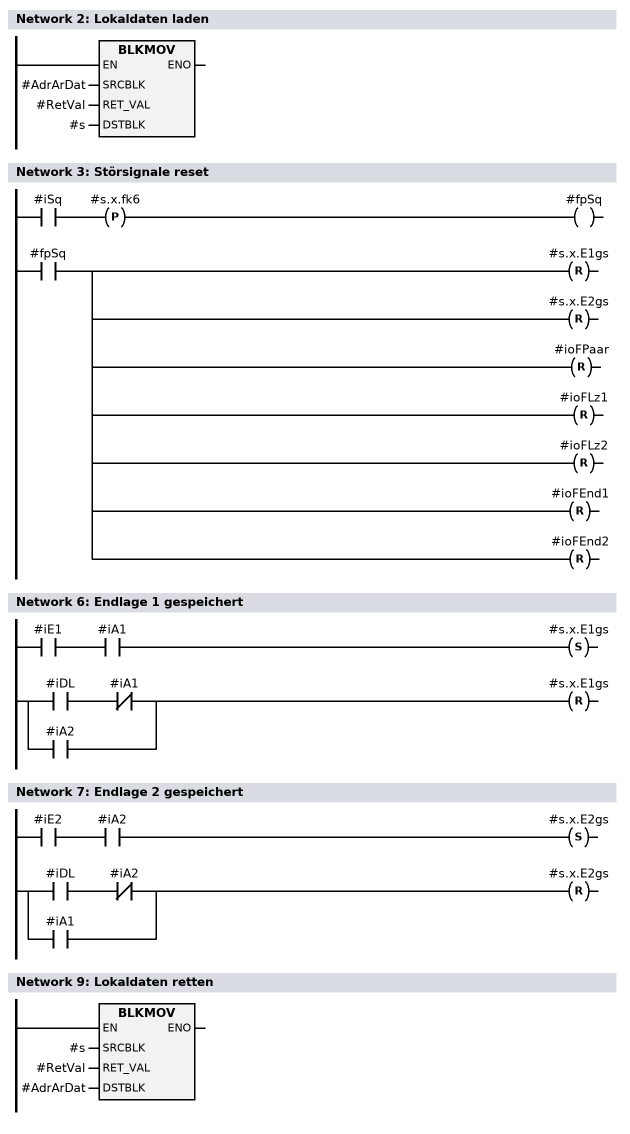
NETWORK
TITLE = Lokaldaten laden
      CALL  "BLKMOV" (
           SRCBLK                   := #AdrArDat,
           RET_VAL                  := #RetVal,
           DSTBLK                   := #s);
      NOP   0;
NETWORK
TITLE = Störsignale reset
      A     #iSq;
      FP    #s.x.fk6;
      =     #fpSq;
      A     #fpSq;
      R     #s.x.E1gs;
      R     #s.x.E2gs;
      R     #ioFPaar;
      R     #ioFLz1;
      R     #ioFLz2;
      R     #ioFEnd1;
      R     #ioFEnd2;
NETWORK
TITLE = Fehler: Paarüberwachung
      L     T#0MS;
      L     #iWPaar;
      ==D;
      O     #iNoPaar;
      JC    t0e1;	//Zeitvorgabe 0ms schaltet Überwachung ab
      R     #seAbgel;
      A     #iE1;
      A     #iE2;
      AN    #fpSq;
      =     #seEingang;
//*** SwZeit ***
      A     #seEingang;
      FP    #s.x.fk0;
      =     #seFpEing;
      AN    #seEingang;
      JC    t0e0;
      L     #iAktTime;
      AN    #seFpEing;
      JC    t0m1;
      T     #s.SwT[0];
t0m1: L     #s.SwT[0];
      -D;
      JPZ   t0m2;
      L     L#2147483647;
      +D;
t0m2: L     #iWPaar;
      >=D;
      =     #seAbgel;
t0e0: A     #seEingang;
      A     #seAbgel;
      =     #seAusgang;
//*** Ende SwZeit ***
      A     #seAusgang;
      S     #ioFPaar;
t0e1: NOP   0;
NETWORK
TITLE = Fehler: Laufzeit
      A     #iA1;
      FP    #s.x.fk4;
      =     #fpiA1;
      A     #iA2;
      FP    #s.x.fk5;
      =     #fpiA2;
      L     T#0MS;
      L     #iWLz;
      ==D;
      O     #iNoLz;
      JC    t1e1;	//Zeitvorgabe 0ms schaltet Überwachung ab
      R     #seAbgel;
      A(;
      AN    #iE1;
      A     #iA1;
      AN    #fpiA1;	//bei direkter Richtungsumschaltung Zeit neu triggern
      AN    #s.x.E1gs;
      O;
      AN    #iE2;
      A     #iA2;
      AN    #fpiA2;	//bei direkter Richtungsumschaltung Zeit neu triggern
      AN    #s.x.E2gs;
      );
      AN    #fpSq;
      =     #seEingang;
//*** SwZeit 1 ***
      A     #seEingang;
      FP    #s.x.fk1;
      =     #seFpEing;
      AN    #seEingang;
      JC    t1e0;
      L     #iAktTime;
      AN    #seFpEing;
      JC    t1m1;
      T     #s.SwT[1];
t1m1: L     #s.SwT[1];
      -D;
      JPZ   t1m2;
      L     L#2147483647;
      +D;
t1m2: L     #iWLz;
      >=D;
      =     #seAbgel;
t1e0: A     #seEingang;
      A     #seAbgel;
      =     #seAusgang;
//*** Ende SwZeit ***
      A     #seAusgang;
      A     #iA1;
      S     #ioFLz1;
      A     #seAusgang;
      A     #iA2;
      S     #ioFLz2;
t1e1: NOP   0;
NETWORK
TITLE = Endlage 1 gespeichert
      A     #iE1;
      A     #iA1;
      S     #s.x.E1gs;
      A(;
      A     #iDL;
      AN    #iA1;
      O     #iA2;
      );
      R     #s.x.E1gs;
      NOP   0;
NETWORK
TITLE = Endlage 2 gespeichert
      A     #iE2;
      A     #iA2;
      S     #s.x.E2gs;
      A(;
      A     #iDL;
      AN    #iA2;
      O     #iA1;
      );
      R     #s.x.E2gs;
      NOP   0;
NETWORK
TITLE = Fehler: Endlage verlassen
      L     T#0MS;
      L     #iWEndl;
      ==D;
      O     #iNoEnd;
      JC    t2e1;	//Zeitvorgabe 0ms schaltet Überwachung ab
      R     #seAbgel;
      A(;
      A     #s.x.E1gs;
      AN    #iE1;
      O;
      A     #s.x.E2gs;
      AN    #iE2;
      );
      AN    #fpSq;
      =     #seEingang;
//*** SwZeit 2 ***
      A     #seEingang;
      FP    #s.x.fk2;
      =     #seFpEing;
      AN    #seEingang;
      JC    t2e0;
      L     #iAktTime;
      AN    #seFpEing;
      JC    t2m1;
      T     #s.SwT[2];
t2m1: L     #s.SwT[2];
      -D;
      JPZ   t2m2;
      L     L#2147483647;
      +D;
t2m2: L     #iWEndl;
      >=D;
      =     #seAbgel;
t2e0: A     #seEingang;
      A     #seAbgel;
      =     #seAusgang;
//*** Ende SwZeit ***
      A     #seAusgang;
      A     #s.x.E1gs;
      AN    #iE1;
      S     #ioFEnd1;
      A     #seAusgang;
      A     #s.x.E2gs;
      AN    #iE2;
      S     #ioFEnd2;
t2e1: NOP   0;
NETWORK
TITLE = Lokaldaten retten
      CALL  "BLKMOV" (
           SRCBLK                   := #s,
           RET_VAL                  := #RetVal,
           DSTBLK                   := #AdrArDat);
      NOP   0;
END_FUNCTION

FUNCTION "FC_CK1OP" : VOID	// FC 102
TITLE = Überwachung von 1 Aus-/Eingang
//________________________________________________________________________________
//$Revision: x.y $
//$Date: 2005/04/26 0:0:0CET $
//$Author: slh $
//$ProjectRevision: Last Checkpoint: m.n $
//
//-------------------------------------------------------------------------------
//*ALL RIGHTS RESERVED
//*Softwareentwicklung
//erstellt: 09.05.2005; Helmut Scheuenstuhl (slh); Scheuenstuhl PAC / V0.1
//Änderung: Datum / Abteilung / Name / Version x.y
//Änderung: 
//        :
//-------------------------------------------------------------------------------
//Beschreibung
//Der Fc dient zur Überwachung von 1 Stellglied (Ventile o.ä.)
//Pro Aufruf werden 14 Byte Arbeitsdaten benötigt, deren Adresse über 
//iArbDat(Any) angegeben wird.
//WICHTIGE VORAUSSETZUNG:
//Der Fc arbeitet mit der Plc-Zeit, die mit SFC64 Time_tck ausgelesen und am
//"iAktTime" angeboten werden muß.
AUTHOR : SPAC_slh
FAMILY : Diagnose
NAME : CK1OP
VERSION : 0.1
VAR_INPUT
  iArbDat : ANY ;	//Rettadresse der 14Byte Arbeitsdaten des Fc
  iAktTime : TIME ;	//ausgeleseneSysZeitVonTime_tck SFC64
  iWAus : TIME ;	//Verzögerung Ausschaltüberwachung, T#0MS= Abwahl
  iWEin : TIME ;	//Verzögerung Einschaltüberwachung, T#0MS= Abwahl
  iWUnt : TIME ;	//Verzögerung Unterbrechungsüberwachung, T#0MS= Abwahl
  iE1 : BOOL ;	//Schalter, wird durch iA1 angefahren
  iA1 : BOOL ;	//zu überwachender Ausgang 1
  iSq : BOOL ;	//Störung quittieren
END_VAR
VAR_IN_OUT
  ioFEin : BOOL ;	//Fehler Einschaltüberwachung
  ioFUnt : BOOL ;	//Fehler:Unterbrechungsüberwachung
  ioFAus : BOOL ;	//Fehler Ausschaltüberwachung
END_VAR
VAR_TEMP
  AdrArDat : ANY ;	//Übergabeparameter für Adresse der Arbeitsdaten
  svAr1 : DWORD ;
  svAr2 : DWORD ;
  s : UDT 1010;	//stat, da gerettet
  RetVal : INT ;
  Lop1 : BOOL ;
  seEingang : BOOL ;	//SwTimer se Eingang
  seFpEing : BOOL ;	//SwTimer se Eingang pos.Flanke
  seAbgel : BOOL ;	//SwTimer se abgelaufen
  seAusgang : BOOL ;	//SwTimer se Ausgang
  fpiA1 : BOOL ;
  fpSq : BOOL ;	//Flanke Störung quittieren
END_VAR
BEGIN
NETWORK
TITLE = Übergabezeiger für BLKMOV aus iArbDat übernehmen
      TAR1  #svAr1;
      TAR2  #svAr2;
      L     P##iArbDat;
      LAR1;
      LAR2  P##AdrArDat;
      L     W [AR1,P#0.0];
      T     LW [AR2,P#0.0];
      L     D [AR1,P#2.0];
      T     LD [AR2,P#2.0];
      L     D [AR1,P#6.0];
      T     LD [AR2,P#6.0];
      LAR1  #svAr1;
      LAR2  #svAr2;
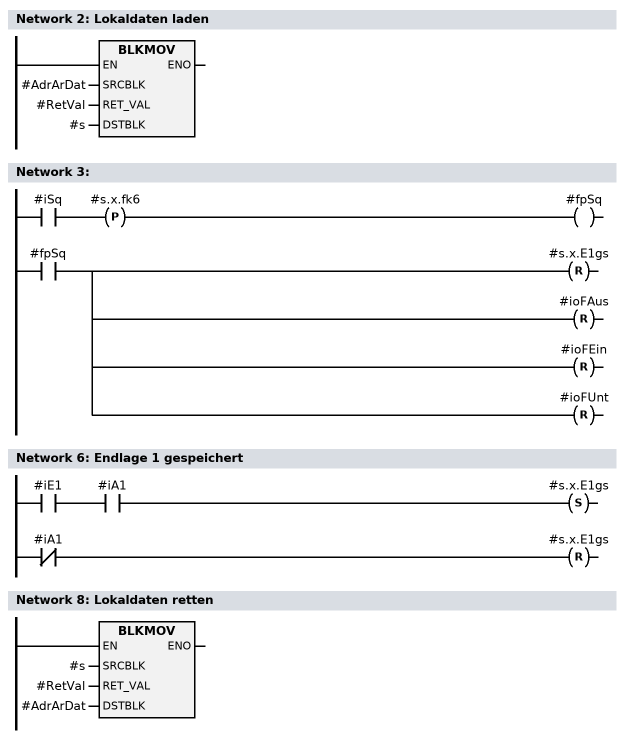
NETWORK
TITLE = Lokaldaten laden
      CALL  "BLKMOV" (
           SRCBLK                   := #AdrArDat,
           RET_VAL                  := #RetVal,
           DSTBLK                   := #s);
      NOP   0;
NETWORK
TITLE =
      A     #iSq;
      FP    #s.x.fk6;
      =     #fpSq;
      A     #fpSq;
      R     #s.x.E1gs;
      R     #ioFAus;
      R     #ioFEin;
      R     #ioFUnt;
NETWORK
TITLE = Fehler: Ausschaltüberwachung
      L     T#0MS;
      L     #iWAus;
      ==D;
      JC    t0e1;	//Zeitvorgabe 0ms schaltet Überwachung ab
      R     #seAbgel;
      A     #iE1;
      AN    #iA1;
      AN    #fpSq;
      =     #seEingang;
//*** SwZeit ***
      A     #seEingang;
      FP    #s.x.fk0;
      =     #seFpEing;
      AN    #seEingang;
      JC    t0e0;
      L     #iAktTime;
      AN    #seFpEing;
      JC    t0m1;
      T     #s.SwT[0];
t0m1: L     #s.SwT[0];
      -D;
      JPZ   t0m2;
      L     L#2147483647;
      +D;
t0m2: L     #iWAus;
      >=D;
      =     #seAbgel;
t0e0: A     #seEingang;
      A     #seAbgel;
      =     #seAusgang;
//*** Ende SwZeit ***
      A     #seAusgang;
      S     #ioFAus;
t0e1: NOP   0;
NETWORK
TITLE = Fehler: Laufzeit, Einschaltüberwachung
      A     #iA1;
      FP    #s.x.fk4;
      =     #fpiA1;
      L     T#0MS;
      L     #iWEin;
      ==D;
      JC    t1e1;	//Zeitvorgabe 0ms schaltet Überwachung ab
      R     #seAbgel;
      AN    #iE1;
      A     #iA1;
      AN    #s.x.E1gs;
      AN    #fpSq;
      =     #seEingang;
//*** SwZeit 1 ***
      A     #seEingang;
      FP    #s.x.fk1;
      =     #seFpEing;
      AN    #seEingang;
      JC    t1e0;
      L     #iAktTime;
      AN    #seFpEing;
      JC    t1m1;
      T     #s.SwT[1];
t1m1: L     #s.SwT[1];
      -D;
      JPZ   t1m2;
      L     L#2147483647;
      +D;
t1m2: L     #iWEin;
      >=D;
      =     #seAbgel;
t1e0: A     #seEingang;
      A     #seAbgel;
      =     #seAusgang;
//*** Ende SwZeit ***
      A     #seAusgang;
      S     #ioFEin;
t1e1: NOP   0;
NETWORK
TITLE = Endlage 1 gespeichert
      A     #iE1;
      A     #iA1;
      S     #s.x.E1gs;
      AN    #iA1;
      R     #s.x.E1gs;
      NOP   0;
NETWORK
TITLE = Fehler: Endlage verlassen=Unterbrechungsüberwachung
      L     T#0MS;
      L     #iWUnt;
      ==D;
      JC    t2e1;	//Zeitvorgabe 0ms schaltet Überwachung ab
      R     #seAbgel;
      A     #s.x.E1gs;
      AN    #iE1;
      AN    #fpSq;
      =     #seEingang;
//*** SwZeit 2 ***
      A     #seEingang;
      FP    #s.x.fk2;
      =     #seFpEing;
      AN    #seEingang;
      JC    t2e0;
      L     #iAktTime;
      AN    #seFpEing;
      JC    t2m1;
      T     #s.SwT[2];
t2m1: L     #s.SwT[2];
      -D;
      JPZ   t2m2;
      L     L#2147483647;
      +D;
t2m2: L     #iWUnt;
      >=D;
      =     #seAbgel;
t2e0: A     #seEingang;
      A     #seAbgel;
      =     #seAusgang;
//*** Ende SwZeit ***
      A     #seAusgang;
      A     #s.x.E1gs;
      AN    #iE1;
      S     #ioFUnt;
t2e1: NOP   0;
NETWORK
TITLE = Lokaldaten retten
      CALL  "BLKMOV" (
           SRCBLK                   := #s,
           RET_VAL                  := #RetVal,
           DSTBLK                   := #AdrArDat);
      NOP   0;
END_FUNCTION

FUNCTION "INPUT_MASTER" : VOID	// FC 111
TITLE = EINGÄNGE VOM MASTERSYSTEM LESEN
//Die Kommunikation mit dem Mastersystem erfolgt durch Merkerwörter
AUTHOR : APetz
VERSION : 0.1
VAR_TEMP
  B_TEMP : BYTE ;	//Zwischenspeicher
  X_TEMP : BOOL ;	//Zwischenspeicher
END_VAR
BEGIN
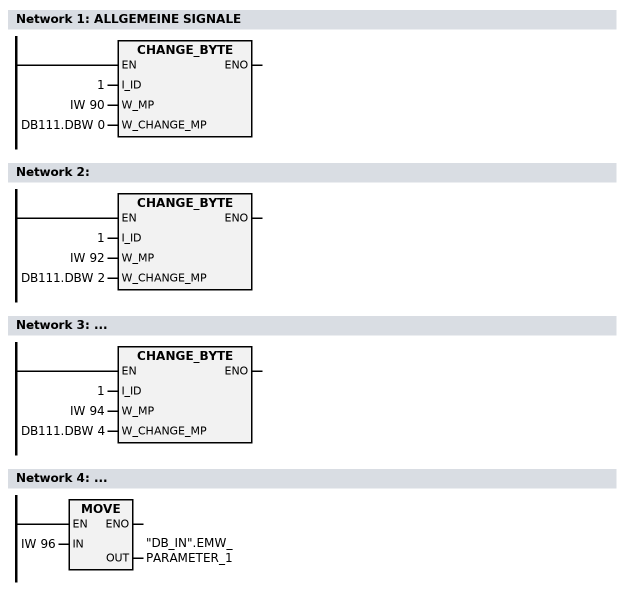
NETWORK
TITLE = ALLGEMEINE SIGNALE
//Eingangswort in Datenbaustein transferieren
//EW90 (aus HW-Konfiguration) nach DB111.DBW0 schreiben (Byte-/Bitzugriff)
//HINWEIS: Das Tauschen der Bytes wird, durch die unterschiedlichen Notationen,
//         benötigt.
      CALL  "CHANGE_BYTE" (
           I_ID                     := 1,
           W_MP                     := IW 90,
           W_CHANGE_MP              := DB111.DBW 0);
      NOP   0;
NETWORK
TITLE =
//Eingangswort in Datenbaustein transferieren
//EW92 (aus HW-Konfiguration) nach DB111.DBW2 schreiben (Byte-/Bitzugriff)
//HINWEIS: Das Tauschen der Bytes wird, durch die unterschiedlichen Notationen,
//         benötigt.
      CALL  "CHANGE_BYTE" (
           I_ID                     := 1,
           W_MP                     := IW 92,
           W_CHANGE_MP              := DB111.DBW 2);
      NOP   0;
NETWORK
TITLE = ...
//Eingangswort in Datenbaustein transferieren
//EW94 (aus HW-Konfiguration) nach DB111.DBW4 schreiben (Byte-/Bitzugriff)
//HINWEIS: Das Tauschen der Bytes wird, durch die unterschiedlichen Notationen,
//         benötigt.
      CALL  "CHANGE_BYTE" (
           I_ID                     := 1,
           W_MP                     := IW 94,
           W_CHANGE_MP              := DB111.DBW 4);
      NOP   0;
NETWORK
TITLE = ...
//Eingangswort in Datenbaustein transferieren
//EW96 (aus HW-Konfiguration) nach DB111.DBW6 schreiben (Byte-/Bitzugriff)
//HINWEIS: Das Tauschen der Bytes wird, durch die unterschiedlichen Notationen,
//         benötigt.
      L     IW 96;
      T     "DB_IN".EMW_PARAMETER_1;
      NOP   0;
END_FUNCTION

FUNCTION "OUTPUT_MASTER" : VOID	// FC 112
TITLE = AUSGÄNGE AN MASTERSYSTEM SCHREIBEN
//Die Kommunikation mit dem Mastersystem erfolgt durch Merkerwörter
AUTHOR : APetz
VERSION : 0.1
BEGIN
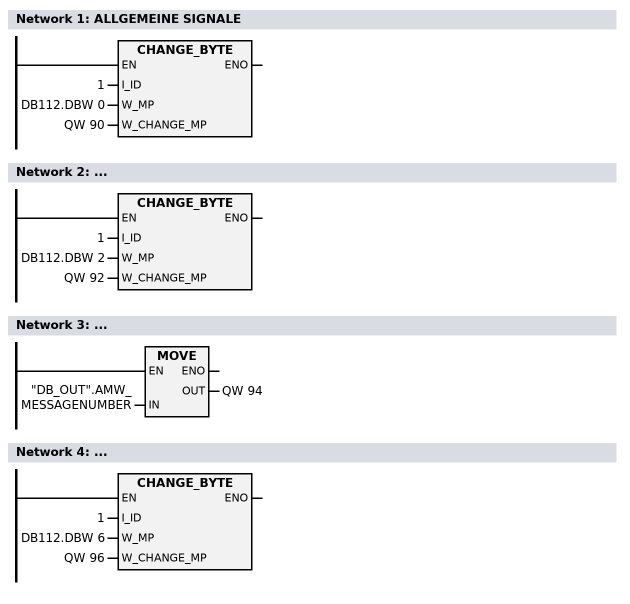
NETWORK
TITLE = ALLGEMEINE SIGNALE
//Datenbaustein nach Ausgangswort transferieren
//DB112.DBW0 nach AW90 (HW-Konfiguration) schreiben (Byte-/Bitzugriff)
//HINWEIS: Das Tauschen der Bytes wird, durch die unterschiedlichen Notationen,
//         benötigt.
      CALL  "CHANGE_BYTE" (
           I_ID                     := 1,
           W_MP                     := DB112.DBW 0,
           W_CHANGE_MP              := QW 90);
      NOP   0;
NETWORK
TITLE = ...
//Datenbaustein nach Ausgangswort transferieren
//DB112.DBW2 nach AW92 (HW-Konfiguration) schreiben (Byte-/Bitzugriff)
//HINWEIS: Das Tauschen der Bytes wird, durch die unterschiedlichen Notationen,
//         benötigt.
      CALL  "CHANGE_BYTE" (
           I_ID                     := 1,
           W_MP                     := DB112.DBW 2,
           W_CHANGE_MP              := QW 92);
      NOP   0;
NETWORK
TITLE = ...
//Datenbaustein nach Ausgangswort transferieren
//DB112.DBW4 nach AW94 (HW-Konfiguration) schreiben (Byte-/Bitzugriff)
//HINWEIS: Das Tauschen der Bytes wird, durch die unterschiedlichen Notationen,
//         benötigt.
      L     "DB_OUT".AMW_MESSAGENUMBER;
      T     QW 94;
      NOP   0;
NETWORK
TITLE = ...
//Datenbaustein nach Ausgangswort transferieren
//DB112.DBW6 nach AW96 (HW-Konfiguration) schreiben (Byte-/Bitzugriff)
//HINWEIS: Das Tauschen der Bytes wird, durch die unterschiedlichen Notationen,
//         benötigt.
      CALL  "CHANGE_BYTE" (
           I_ID                     := 1,
           W_MP                     := DB112.DBW 6,
           W_CHANGE_MP              := QW 96);
      NOP   0;
END_FUNCTION

FUNCTION "INPUT_PERIPHERIE" : VOID	// FC 121
TITLE = EINGÄNGE VOM PERPHERIE LESEN
//Eingangssignale von Peripherie (ET200S) rangieren
AUTHOR : APetz
VERSION : 0.1
VAR_TEMP
  B_TEMP : BYTE ;	//Zwischenspeicher
  X_TEMP : BOOL ;	//Zwischenspeicher
  TMP_BIT_ENABLE : BOOL ;	//Bausteinfreigabe - Sammelstörung
END_VAR
BEGIN
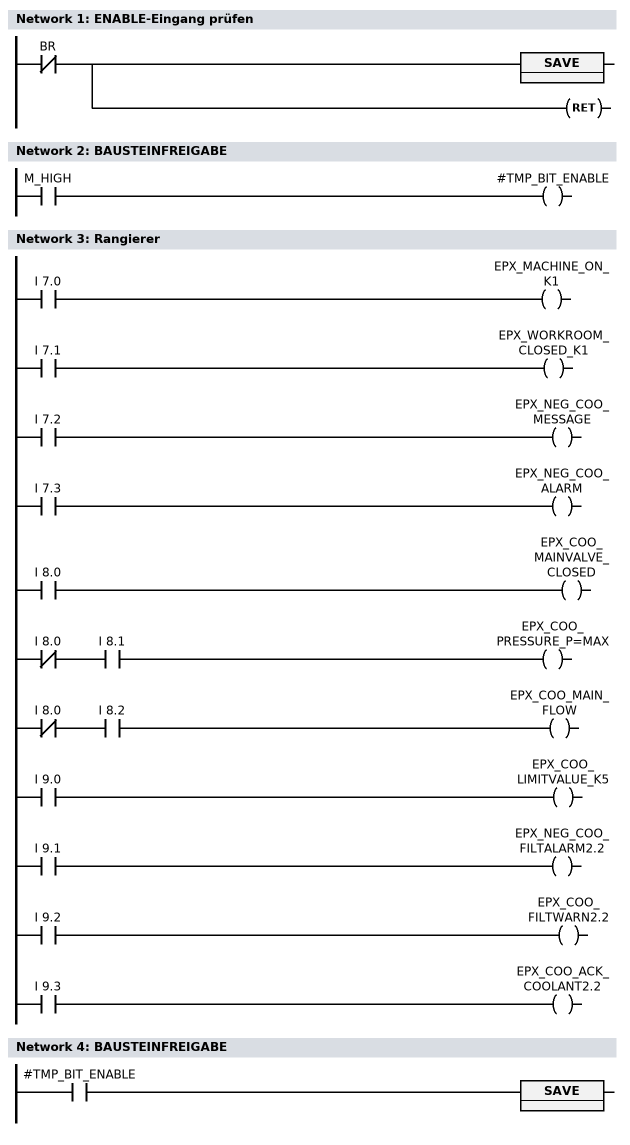
NETWORK
TITLE = ENABLE-Eingang prüfen
//Auswerten des BIE-Statusbit. Dieses entspricht dem EN (ENABLE)-Einganges bei 
//KOP/FUP. Wenn EN=FALSE dann verlasse Baustein.
//
      AN    BR;
      SAVE;
      BEC;
NETWORK
TITLE = BAUSTEINFREIGABE
//Fehlerauswertung Baustein intern:
//Bausteinfreigabe wird gesetzt
      A     "M_HIGH";
      =     #TMP_BIT_ENABLE;
NETWORK
TITLE = Rangierer
      A     I 7.0;
      =     "EPX_MACHINE_ON_K1";
      A     I 7.1;
      =     "EPX_WORKROOM_CLOSED_K1";
      A     I 7.2;
      =     "EPX_NEG_COO_MESSAGE";
      A     I 7.3;
      =     "EPX_NEG_COO_ALARM";
      A     I 8.0;
      =     "EPX_COO_MAINVALVE_CLOSED";
      AN    I 8.0;
      A     I 8.1;
      =     "EPX_COO_PRESSURE_P=MAX";
      AN    I 8.0;
      A     I 8.2;
      =     "EPX_COO_MAIN_FLOW";
      A     I 9.0;
      =     "EPX_COO_LIMITVALUE_K5";
      A     I 9.1;
      =     "EPX_NEG_COO_FILTALARM2.2";
      A     I 9.2;
      =     "EPX_COO_FILTWARN2.2";
      A     I 9.3;
      =     "EPX_COO_ACK_COOLANT2.2";
NETWORK
TITLE = BAUSTEINFREIGABE
//Statusbit BIE=ENO setzen, wenn Funktion ohne Fehler durchlaufen wurde.
      A     #TMP_BIT_ENABLE;
      SAVE;
END_FUNCTION

FUNCTION "OUTPUT_PERIPHERIE" : VOID	// FC 122
TITLE = AUSGÄNGE AN PERIPHERIE SCHREIBEN
//Ausgangssignale an Peripherie (ET200S) rangieren
AUTHOR : APetz
VERSION : 0.1
VAR_TEMP
  TMP_BIT_ENABLE : BOOL ;	//Bausteinfreigabe - Sammelstörung
END_VAR
BEGIN
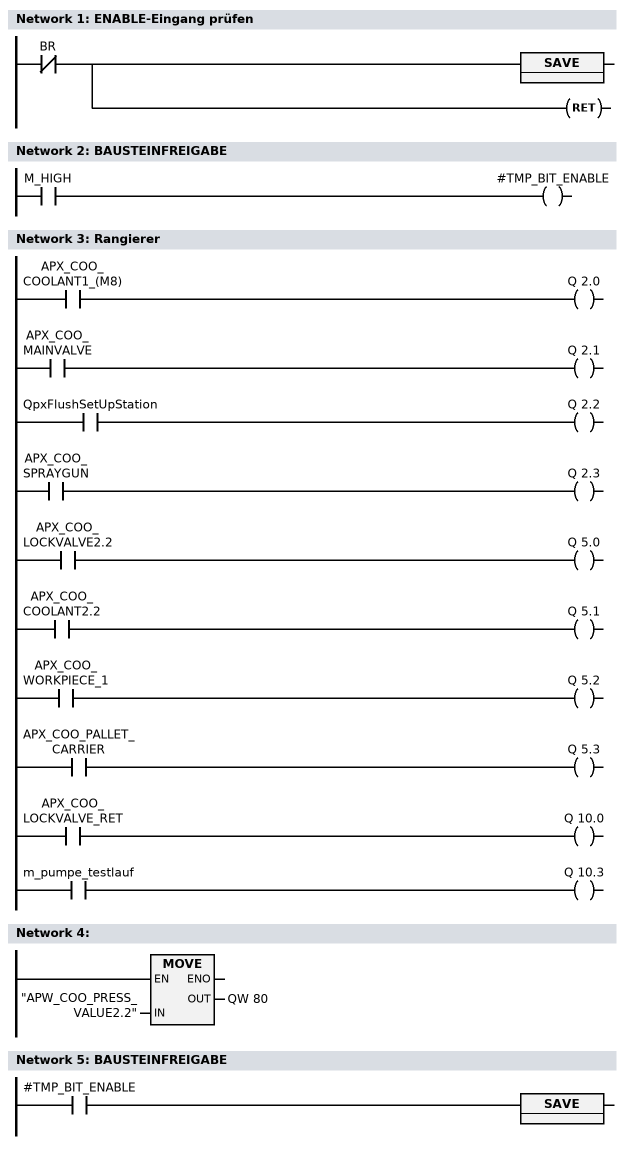
NETWORK
TITLE = ENABLE-Eingang prüfen
//Auswerten des BIE-Statusbit. Dieses entspricht dem EN (ENABLE)-Einganges bei 
//KOP/FUP. Wenn EN=FALSE dann verlasse Baustein.
//
      AN    BR;
      SAVE;
      BEC;
NETWORK
TITLE = BAUSTEINFREIGABE
//Fehlerauswertung Baustein intern:
//Bausteinfreigabe wird gesetzt
      A     "M_HIGH";
      =     #TMP_BIT_ENABLE;
NETWORK
TITLE = Rangierer
      A     "APX_COO_COOLANT1_(M8)";
      =     Q 2.0;
      A     "APX_COO_MAINVALVE";
      =     Q 2.1;
      A     "QpxFlushSetUpStation";
      =     Q 2.2;
      A     "APX_COO_SPRAYGUN";
      =     Q 2.3;
      A     "APX_COO_LOCKVALVE2.2";
      =     Q 5.0;
      A     "APX_COO_COOLANT2.2";
      =     Q 5.1;
      A     "APX_COO_WORKPIECE_1";
      =     Q 5.2;
      A     "APX_COO_PALLET_CARRIER";
      =     Q 5.3;
      A     "APX_COO_LOCKVALVE_RET";
      =     Q 10.0;
// zur Steuerung der Versorgungspumpe auf
// dem hausinternen Teststand (=Testlauf)
      A     "m_pumpe_testlauf";
      =     Q 10.3;
NETWORK
TITLE =
//Rangierer für Analogbaugruppe
      L     "APW_COO_PRESS_VALUE2.2";
      T     QW 80;
      NOP   0;
NETWORK
TITLE = BAUSTEINFREIGABE
//Statusbit BIE=ENO setzen, wenn Funktion ohne Fehler durchlaufen wurde.
      A     #TMP_BIT_ENABLE;
      SAVE;
END_FUNCTION

DATA_BLOCK "DB_MESSAGE"	// DB 2
AUTHOR : SPAC_slh
VERSION : 0.1
  STRUCT
   ALARM_001 : BOOL ;	//Schaltschranktemperatur zu hoch
   ALARM_002 : BOOL ;	//Schaltschranktemperatur - Grenzwert überschritten
   F003 : BOOL ;	//1-
   F004 : BOOL ;	//1-
   F005 : BOOL ;	//1-
   F006 : BOOL ;	//1-
   F007 : BOOL ;	//1-
   F008 : BOOL ;	//1-
   F009 : BOOL ;	//1-
   F010 : BOOL ;	//1-
   F011 : BOOL ;	//1-
   F012 : BOOL ;	//1-
   F013 : BOOL ;	//1-
   F014 : BOOL ;	//1-
   F015 : BOOL ;	//1-
   F016 : BOOL ;	//1-
   F017 : BOOL ;	//Spanner 1 LzFehler lösen
   F018 : BOOL ;	//Spanner 1 LzFehler spannen
   F019 : BOOL ;	//Spanner 1 Fehler Endlage gelöst
   F020 : BOOL ;	//Spanner 1 Fehler Endlage gespannt
   F021 : BOOL ;	//Spanner 1 Fehler Paarüberwachung
   F022 : BOOL ;	//Spanner 2 LzFehler lösen
   F023 : BOOL ;	//Spanner 2 LzFehler spannen
   F024 : BOOL ;	//Spanner 2 Fehler Endlage gelöst
   F025 : BOOL ;	//Spanner 2 Fehler Endlage gespannt
   F026 : BOOL ;	//Spanner 2 Fehler Paarüberwachung
   F027 : BOOL ;	//Auflagektrl.LzFehler bei einschalten
   F028 : BOOL ;	//Auflagektrl.LzFehler bei ausschalten
   F029 : BOOL ;	//Auflagektrl.Fehler Endlage Druck erreicht
   F030 : BOOL ;	//Auflagektrl.Fehler Endlage Drucklos
   F031 : BOOL ;	//Auflagektrl.Fehler Paarüberwachung
   F032 : BOOL ;	//Verriegelungsktrl.LzFehler bei einschalten
   F033 : BOOL ;	//Verriegelungsktrl.LzFehler bei ausschalten
   F034 : BOOL ;	//Verriegelungsktrl.Fehler Endlage Druck erreicht
   F035 : BOOL ;	//Verriegelungsktrl.Fehler Endlage Drucklos
   F036 : BOOL ;	//Verriegelungsktrl.Fehler Paarüberwachung
   F037 : BOOL ;	//1-
   F038 : BOOL ;	//1-
   F039 : BOOL ;	//1-
   F040 : BOOL ;	//1-
   F041 : BOOL ;	//1-
   F042 : BOOL ;	//1-
   F043 : BOOL ;	//1-
   F044 : BOOL ;	//1-
   F045 : BOOL ;	//1-
   F046 : BOOL ;	//1-
   F047 : BOOL ;	//1-
   F048 : BOOL ;	//1-
   F049 : BOOL ;	//1-
   F050 : BOOL ;	//1-
   F051 : BOOL ;	//1-
   F052 : BOOL ;	//1-
   F053 : BOOL ;	//1-
   F054 : BOOL ;	//1-
   F055 : BOOL ;	//1-
   F056 : BOOL ;	//1-
   F057 : BOOL ;	//1-
   F058 : BOOL ;	//1-
   F059 : BOOL ;	//1-
   F060 : BOOL ;	//1-
   F061 : BOOL ;	//1-
   F062 : BOOL ;	//1-
   F063 : BOOL ;	//1-
   F064 : BOOL ;	//1-
   F065 : BOOL ;	//1-
   F066 : BOOL ;	//1-
   F067 : BOOL ;	//1-
   F068 : BOOL ;	//1-
   F069 : BOOL ;	//1-
   F070 : BOOL ;	//1-
   F071 : BOOL ;	//1-
   F072 : BOOL ;	//1-
   F073 : BOOL ;	//1-
   F074 : BOOL ;	//1-
   F075 : BOOL ;	//1-
   F076 : BOOL ;	//1-
   F077 : BOOL ;	//1-
   F078 : BOOL ;	//1-
   F079 : BOOL ;	//1-
   F080 : BOOL ;	//1-
   F081 : BOOL ;	//1-
   F082 : BOOL ;	//1-
   F083 : BOOL ;	//1-
   F084 : BOOL ;	//1-
   F085 : BOOL ;	//1-
   F086 : BOOL ;	//1-
   F087 : BOOL ;	//1-
   F088 : BOOL ;	//1-
   F089 : BOOL ;	//1-
   F090 : BOOL ;	//1-
   F091 : BOOL ;	//1-
   F092 : BOOL ;	//1-
   F093 : BOOL ;	//1-
   F094 : BOOL ;	//1-
   F095 : BOOL ;	//1-
   F096 : BOOL ;	//1-
   F097 : BOOL ;	//1-
   F098 : BOOL ;	//1-
   F099 : BOOL ;	//1-
   F100 : BOOL ;	//1-
   F101 : BOOL ;	//1-
   F102 : BOOL ;	//1-
   F103 : BOOL ;	//1-
   F104 : BOOL ;	//1-
   F105 : BOOL ;	//1-
   F106 : BOOL ;	//1-
   F107 : BOOL ;	//1-
   F108 : BOOL ;	//1-
   F109 : BOOL ;	//1-
   F110 : BOOL ;	//1-
   F111 : BOOL ;	//1-
   F112 : BOOL ;	//1-
   F113 : BOOL ;	//1-
   F114 : BOOL ;	//1-
   F115 : BOOL ;	//1-
   F116 : BOOL ;	//1-
   F117 : BOOL ;	//1-
   F118 : BOOL ;	//1-
   F119 : BOOL ;	//1-
   F120 : BOOL ;	//1-
   F121 : BOOL ;	//1-
   F122 : BOOL ;	//1-
   F123 : BOOL ;	//1-
   F124 : BOOL ;	//1-
   F125 : BOOL ;	//1-
   F126 : BOOL ;	//1-
   F127 : BOOL ;	//1-
   F128 : BOOL ;	//1-
   F129 : BOOL ;	//1-
   F130 : BOOL ;	//1-
   F131 : BOOL ;	//1-
   F132 : BOOL ;	//1-
   F133 : BOOL ;	//1-
   F134 : BOOL ;	//1-
   F135 : BOOL ;	//1-
   F136 : BOOL ;	//1-
   F137 : BOOL ;	//1-
   F138 : BOOL ;	//1-
   F139 : BOOL ;	//1-
   F140 : BOOL ;	//1-
   F141 : BOOL ;	//1-
   F142 : BOOL ;	//1-
   F143 : BOOL ;	//1-
   F144 : BOOL ;	//1-
   F145 : BOOL ;	//1-
   F146 : BOOL ;	//1-
   F147 : BOOL ;	//1-
   F148 : BOOL ;	//1-
   F149 : BOOL ;	//1-
   F150 : BOOL ;	//1-
   F151 : BOOL ;	//1-
   F152 : BOOL ;	//1-
   F153 : BOOL ;	//1-
   F154 : BOOL ;	//1-
   F155 : BOOL ;	//1-
   F156 : BOOL ;	//1-
   F157 : BOOL ;	//1-
   F158 : BOOL ;	//1-
   F159 : BOOL ;	//1-
   F160 : BOOL ;	//1-
   F161 : BOOL ;	//1-
   F162 : BOOL ;	//1-
   F163 : BOOL ;	//1-
   F164 : BOOL ;	//1-
   F165 : BOOL ;	//1-
   F166 : BOOL ;	//1-
   F167 : BOOL ;	//1-
   F168 : BOOL ;	//1-
   F169 : BOOL ;	//1-
   F170 : BOOL ;	//1-
   F171 : BOOL ;	//1-
   F172 : BOOL ;	//1-
   F173 : BOOL ;	//1-
   F174 : BOOL ;	//1-
   F175 : BOOL ;	//1-
   F176 : BOOL ;	//1-
   F177 : BOOL ;	//1-
   F178 : BOOL ;	//1-
   F179 : BOOL ;	//1-
   F180 : BOOL ;	//1-
   F181 : BOOL ;	//1-
   F182 : BOOL ;	//1-
   F183 : BOOL ;	//1-
   F184 : BOOL ;	//1-
   F185 : BOOL ;	//1-
   F186 : BOOL ;	//1-
   F187 : BOOL ;	//1-
   F188 : BOOL ;	//1-
   F189 : BOOL ;	//1-
   F190 : BOOL ;	//1-
   F191 : BOOL ;	//1-
   F192 : BOOL ;	//1-
   F193 : BOOL ;	//1-
   F194 : BOOL ;	//1-
   F195 : BOOL ;	//1-
   F196 : BOOL ;	//1-
   F197 : BOOL ;	//1-
   F198 : BOOL ;	//1-
   F199 : BOOL ;	//1-
   F200 : BOOL ;	//1-
   F201 : BOOL ;	//1-
   F202 : BOOL ;	//1-
   F203 : BOOL ;	//1-
   F204 : BOOL ;	//1-
   F205 : BOOL ;	//1-
   F206 : BOOL ;	//1-
   F207 : BOOL ;	//1-
   F208 : BOOL ;	//1-
   F209 : BOOL ;	//1-
   F210 : BOOL ;	//1-
   F211 : BOOL ;	//1-
   F212 : BOOL ;	//1-
   F213 : BOOL ;	//1-
   F214 : BOOL ;	//1-
   F215 : BOOL ;	//1-
   F216 : BOOL ;	//1-
   F217 : BOOL ;	//1-
   F218 : BOOL ;	//1-
   F219 : BOOL ;	//1-
   F220 : BOOL ;	//1-
   F221 : BOOL ;	//1-
   F222 : BOOL ;	//1-
   F223 : BOOL ;	//1-
   F224 : BOOL ;	//1-
   F225 : BOOL ;	//1-
   F226 : BOOL ;	//1-
   F227 : BOOL ;	//1-
   F228 : BOOL ;	//1-
   F229 : BOOL ;	//1-
   F230 : BOOL ;	//1-
   F231 : BOOL ;	//1-
   F232 : BOOL ;	//1-
   F233 : BOOL ;	//1-
   F234 : BOOL ;	//1-
   F235 : BOOL ;	//1-
   F236 : BOOL ;	//1-
   F237 : BOOL ;	//1-
   F238 : BOOL ;	//1-
   F239 : BOOL ;	//1-
   F240 : BOOL ;	//1-
   F241 : BOOL ;	//1-
   F242 : BOOL ;	//1-
   F243 : BOOL ;	//1-
   F244 : BOOL ;	//1-
   F245 : BOOL ;	//1-
   F246 : BOOL ;	//1-
   F247 : BOOL ;	//1-
   F248 : BOOL ;	//1-
   F249 : BOOL ;	//1-
   F250 : BOOL ;	//1-
   F251 : BOOL ;	//1-
   F252 : BOOL ;	//1-
   F253 : BOOL ;	//1-
   F254 : BOOL ;	//1-
   F255 : BOOL ;	//1-
   F256 : BOOL ;	//1-
   F257 : BOOL ;	//1-
   F258 : BOOL ;	//1-
   F259 : BOOL ;	//1-
   F260 : BOOL ;	//1-
   F261 : BOOL ;	//1-
   F262 : BOOL ;	//1-
   F263 : BOOL ;	//1-
   F264 : BOOL ;	//1-
   F265 : BOOL ;	//1-
   F266 : BOOL ;	//1-
   F267 : BOOL ;	//1-
   F268 : BOOL ;	//1-
   F269 : BOOL ;	//1-
   F270 : BOOL ;	//1-
   F271 : BOOL ;	//1-
   F272 : BOOL ;	//1-
   F273 : BOOL ;	//1-
   F274 : BOOL ;	//1-
   F275 : BOOL ;	//1-
   F276 : BOOL ;	//1-
   F277 : BOOL ;	//1-
   F278 : BOOL ;	//1-
   F279 : BOOL ;	//1-
   F280 : BOOL ;	//1-
   F281 : BOOL ;	//1-
   F282 : BOOL ;	//1-
   F283 : BOOL ;	//1-
   F284 : BOOL ;	//1-
   F285 : BOOL ;	//1-
   F286 : BOOL ;	//1-
   F287 : BOOL ;	//1-
   F288 : BOOL ;	//1-
   F289 : BOOL ;	//1-
   F290 : BOOL ;	//1-
   F291 : BOOL ;	//1-
   F292 : BOOL ;	//1-
   F293 : BOOL ;	//1-
   F294 : BOOL ;	//1-
   F295 : BOOL ;	//1-
   F296 : BOOL ;	//1-
   F297 : BOOL ;	//1-
   F298 : BOOL ;	//1-
   F299 : BOOL ;	//1-
   F300 : BOOL ;	//1-
   F301 : BOOL ;	//1-
   F302 : BOOL ;	//1-
   F303 : BOOL ;	//1-
   F304 : BOOL ;	//1-
   F305 : BOOL ;	//1-
   F306 : BOOL ;	//1-
   F307 : BOOL ;	//1-
   F308 : BOOL ;	//1-
   F309 : BOOL ;	//1-
   F310 : BOOL ;	//1-
   F311 : BOOL ;	//1-
   F312 : BOOL ;	//1-
   F313 : BOOL ;	//1-
   F314 : BOOL ;	//1-
   F315 : BOOL ;	//1-
   F316 : BOOL ;	//1-
   F317 : BOOL ;	//1-
   F318 : BOOL ;	//1-
   F319 : BOOL ;	//1-
   F320 : BOOL ;	//1-
   F321 : BOOL ;	//1-
   F322 : BOOL ;	//1-
   F323 : BOOL ;	//1-
   F324 : BOOL ;	//1-
   F325 : BOOL ;	//1-
   F326 : BOOL ;	//1-
   F327 : BOOL ;	//1-
   F328 : BOOL ;	//1-
   F329 : BOOL ;	//1-
   F330 : BOOL ;	//1-
   F331 : BOOL ;	//1-
   F332 : BOOL ;	//1-
   F333 : BOOL ;	//1-
   F334 : BOOL ;	//1-
   F335 : BOOL ;	//1-
   F336 : BOOL ;	//1-
   F337 : BOOL ;	//1-
   F338 : BOOL ;	//1-
   F339 : BOOL ;	//1-
   F340 : BOOL ;	//1-
   F341 : BOOL ;	//1-
   F342 : BOOL ;	//1-
   F343 : BOOL ;	//1-
   F344 : BOOL ;	//1-
   F345 : BOOL ;	//1-
   F346 : BOOL ;	//1-
   F347 : BOOL ;	//1-
   F348 : BOOL ;	//1-
   F349 : BOOL ;	//1-
   F350 : BOOL ;	//1-
   F351 : BOOL ;	//1-
   F352 : BOOL ;	//1-
   F353 : BOOL ;	//1-
   F354 : BOOL ;	//1-
   F355 : BOOL ;	//1-
   F356 : BOOL ;	//1-
   F357 : BOOL ;	//1-
   F358 : BOOL ;	//1-
   F359 : BOOL ;	//1-
   F360 : BOOL ;	//1-
   F361 : BOOL ;	//1-
   F362 : BOOL ;	//1-
   F363 : BOOL ;	//1-
   F364 : BOOL ;	//1-
   F365 : BOOL ;	//1-
   F366 : BOOL ;	//1-
   F367 : BOOL ;	//1-
   F368 : BOOL ;	//1-
   F369 : BOOL ;	//1-
   F370 : BOOL ;	//1-
   F371 : BOOL ;	//1-
   F372 : BOOL ;	//1-
   F373 : BOOL ;	//1-
   F374 : BOOL ;	//1-
   F375 : BOOL ;	//1-
   F376 : BOOL ;	//1-
   F377 : BOOL ;	//1-
   F378 : BOOL ;	//1-
   F379 : BOOL ;	//1-
   F380 : BOOL ;	//1-
   F381 : BOOL ;	//1-
   F382 : BOOL ;	//1-
   F383 : BOOL ;	//1-
   F384 : BOOL ;	//1-
   F385 : BOOL ;	//1-
   F386 : BOOL ;	//1-
   F387 : BOOL ;	//1-
   F388 : BOOL ;	//1-
   F389 : BOOL ;	//1-
   F390 : BOOL ;	//1-
   F391 : BOOL ;	//1-
   F392 : BOOL ;	//1-
   F393 : BOOL ;	//1-
   F394 : BOOL ;	//1-
   F395 : BOOL ;	//1-
   F396 : BOOL ;	//1-
   F397 : BOOL ;	//1-
   F398 : BOOL ;	//1-
   F399 : BOOL ;	//1-
   F400 : BOOL ;	//1-
   F401 : BOOL ;	//1-
   F402 : BOOL ;	//1-
   F403 : BOOL ;	//1-
   F404 : BOOL ;	//1-
   F405 : BOOL ;	//1-
   F406 : BOOL ;	//1-
   F407 : BOOL ;	//1-
   F408 : BOOL ;	//1-
   F409 : BOOL ;	//1-
   F410 : BOOL ;	//1-
   F411 : BOOL ;	//1-
   F412 : BOOL ;	//1-
   F413 : BOOL ;	//1-
   F414 : BOOL ;	//1-
   F415 : BOOL ;	//1-
   F416 : BOOL ;	//1-
   F417 : BOOL ;	//1-
   F418 : BOOL ;	//1-
   F419 : BOOL ;	//1-
   F420 : BOOL ;	//1-
   F421 : BOOL ;	//1-
   F422 : BOOL ;	//1-
   F423 : BOOL ;	//1-
   F424 : BOOL ;	//1-
   F425 : BOOL ;	//1-
   F426 : BOOL ;	//1-
   F427 : BOOL ;	//1-
   F428 : BOOL ;	//1-
   F429 : BOOL ;	//1-
   F430 : BOOL ;	//1-
   F431 : BOOL ;	//1-
   F432 : BOOL ;	//1-
   F433 : BOOL ;	//1-
   F434 : BOOL ;	//1-
   F435 : BOOL ;	//1-
   F436 : BOOL ;	//1-
   F437 : BOOL ;	//1-
   F438 : BOOL ;	//1-
   F439 : BOOL ;	//1-
   F440 : BOOL ;	//1-
   F441 : BOOL ;	//1-
   F442 : BOOL ;	//1-
   F443 : BOOL ;	//1-
   F444 : BOOL ;	//1-
   F445 : BOOL ;	//1-
   F446 : BOOL ;	//1-
   F447 : BOOL ;	//1-
   F448 : BOOL ;	//1-
   F449 : BOOL ;	//1-
   F450 : BOOL ;	//1-
   F451 : BOOL ;	//1-
   F452 : BOOL ;	//1-
   F453 : BOOL ;	//1-
   F454 : BOOL ;	//1-
   F455 : BOOL ;	//1-
   F456 : BOOL ;	//1-
   F457 : BOOL ;	//1-
   F458 : BOOL ;	//1-
   F459 : BOOL ;	//1-
   F460 : BOOL ;	//1-
   F461 : BOOL ;	//1-
   F462 : BOOL ;	//1-
   F463 : BOOL ;	//1-
   F464 : BOOL ;	//1-
   F465 : BOOL ;	//1-
   F466 : BOOL ;	//1-
   F467 : BOOL ;	//1-
   F468 : BOOL ;	//1-
   F469 : BOOL ;	//1-
   F470 : BOOL ;	//1-
   F471 : BOOL ;	//1-
   F472 : BOOL ;	//1-
   F473 : BOOL ;	//1-
   F474 : BOOL ;	//1-
   F475 : BOOL ;	//1-
   F476 : BOOL ;	//1-
   F477 : BOOL ;	//1-
   F478 : BOOL ;	//1-
   F479 : BOOL ;	//1-
   F480 : BOOL ;	//1-
   F481 : BOOL ;	//1-
   F482 : BOOL ;	//1-
   F483 : BOOL ;	//1-
   F484 : BOOL ;	//1-
   F485 : BOOL ;	//1-
   F486 : BOOL ;	//1-
   F487 : BOOL ;	//1-
   F488 : BOOL ;	//1-
   F489 : BOOL ;	//1-
   F490 : BOOL ;	//1-
   F491 : BOOL ;	//1-
   F492 : BOOL ;	//1-
   F493 : BOOL ;	//1-
   F494 : BOOL ;	//1-
   F495 : BOOL ;	//1-
   F496 : BOOL ;	//1-
   F497 : BOOL ;	//1-
   F498 : BOOL ;	//1-
   F499 : BOOL ;	//1-
   F500 : BOOL ;	//1-
   F501 : BOOL ;	//1-
   F502 : BOOL ;	//1-
   F503 : BOOL ;	//1-
   F504 : BOOL ;	//1-
   F505 : BOOL ;	//1-
   F506 : BOOL ;	//1-
   F507 : BOOL ;	//1-
   F508 : BOOL ;	//1-
   F509 : BOOL ;	//1-
   F510 : BOOL ;	//1-
   F511 : BOOL ;	//1-
   F512 : BOOL ;	//1-
   MSG_513 : BOOL ;	//Schaltschranktüre(n) an Werkzeugmaschine geöffnet
   MSG_514 : BOOL ;	//Schaltschranktüre(n) an Kühlschmierstoffanlage geöffnet
   MSG_515 : BOOL ;	//Schaltschranktemperatur zu hoch
   Me516 : BOOL ;	//1-
   Me517 : BOOL ;	//1-
   Me518 : BOOL ;	//1-
   Me519 : BOOL ;	//1-
   Me520 : BOOL ;	//1-
   Me521 : BOOL ;	//1-
   Me522 : BOOL ;	//1-
   Me523 : BOOL ;	//1-
   Me524 : BOOL ;	//1-
   Me525 : BOOL ;	//1-
   Me526 : BOOL ;	//1-
   Me527 : BOOL ;	//1-
   Me528 : BOOL ;	//1-
   Me529 : BOOL ;	//1-
   Me530 : BOOL ;	//1-
   Me531 : BOOL ;	//1-
   Me532 : BOOL ;	//1-
   Me533 : BOOL ;	//1-
   Me534 : BOOL ;	//1-
   Me535 : BOOL ;	//1-
   Me536 : BOOL ;	//1-
   Me537 : BOOL ;	//1-
   Me538 : BOOL ;	//1-
   Me539 : BOOL ;	//1-
   Me540 : BOOL ;	//1-
   Me541 : BOOL ;	//1-
   Me542 : BOOL ;	//1-
   Me543 : BOOL ;	//1-
   Me544 : BOOL ;	//1-
   Me545 : BOOL ;	//1-
   Me546 : BOOL ;	//1-
   Me547 : BOOL ;	//1-
   Me548 : BOOL ;	//1-
   Me549 : BOOL ;	//1-
   Me550 : BOOL ;	//1-
   Me551 : BOOL ;	//1-
   Me552 : BOOL ;	//1-
   Me553 : BOOL ;	//1-
   Me554 : BOOL ;	//1-
   Me555 : BOOL ;	//1-
   Me556 : BOOL ;	//1-
   Me557 : BOOL ;	//1-
   Me558 : BOOL ;	//1-
   Me559 : BOOL ;	//1-
   Me560 : BOOL ;	//1-
   Me561 : BOOL ;	//1-
   Me562 : BOOL ;	//1-
   Me563 : BOOL ;	//1-
   Me564 : BOOL ;	//1-
   Me565 : BOOL ;	//1-
   Me566 : BOOL ;	//1-
   Me567 : BOOL ;	//1-
   Me568 : BOOL ;	//1-
   Me569 : BOOL ;	//1-
   Me570 : BOOL ;	//1-
   Me571 : BOOL ;	//1-
   Me572 : BOOL ;	//1-
   Me573 : BOOL ;	//1-
   Me574 : BOOL ;	//1-
   Me575 : BOOL ;	//1-
   Me576 : BOOL ;	//1-
   Me577 : BOOL ;	//1-
   Me578 : BOOL ;	//1-
   Me579 : BOOL ;	//1-
   Me580 : BOOL ;	//1-
   Me581 : BOOL ;	//1-
   Me582 : BOOL ;	//1-
   Me583 : BOOL ;	//1-
   Me584 : BOOL ;	//1-
   Me585 : BOOL ;	//1-
   Me586 : BOOL ;	//1-
   Me587 : BOOL ;	//1-
   Me588 : BOOL ;	//1-
   Me589 : BOOL ;	//1-
   Me590 : BOOL ;	//1-
   Me591 : BOOL ;	//1-
   Me592 : BOOL ;	//1-
   Me593 : BOOL ;	//1-
   Me594 : BOOL ;	//1-
   Me595 : BOOL ;	//1-
   Me596 : BOOL ;	//1-
   Me597 : BOOL ;	//1-
   Me598 : BOOL ;	//1-
   Me599 : BOOL ;	//1-
   Me600 : BOOL ;	//1-
   Me601 : BOOL ;	//1-
   Me602 : BOOL ;	//1-
   Me603 : BOOL ;	//1-
   Me604 : BOOL ;	//1-
   Me605 : BOOL ;	//1-
   Me606 : BOOL ;	//1-
   Me607 : BOOL ;	//1-
   Me608 : BOOL ;	//1-
   Me609 : BOOL ;	//1-
   Me610 : BOOL ;	//1-
   Me611 : BOOL ;	//1-
   Me612 : BOOL ;	//1-
   Me613 : BOOL ;	//1-
   Me614 : BOOL ;	//1-
   Me615 : BOOL ;	//1-
   Me616 : BOOL ;	//1-
   Me617 : BOOL ;	//1-
   Me618 : BOOL ;	//1-
   Me619 : BOOL ;	//1-
   Me620 : BOOL ;	//1-
   Me621 : BOOL ;	//1-
   Me622 : BOOL ;	//1-
   Me623 : BOOL ;	//1-
   Me624 : BOOL ;	//1-
   Me625 : BOOL ;	//1-
   Me626 : BOOL ;	//1-
   Me627 : BOOL ;	//1-
   Me628 : BOOL ;	//1-
   Me629 : BOOL ;	//1-
   Me630 : BOOL ;	//1-
   Me631 : BOOL ;	//1-
   Me632 : BOOL ;	//1-
   Me633 : BOOL ;	//1-
   Me634 : BOOL ;	//1-
   Me635 : BOOL ;	//1-
   Me636 : BOOL ;	//1-
   Me637 : BOOL ;	//1-
   Me638 : BOOL ;	//1-
   Me639 : BOOL ;	//1-
   Me640 : BOOL ;	//1-
   Me641 : BOOL ;	//1-
   Me642 : BOOL ;	//1-
   Me643 : BOOL ;	//1-
   Me644 : BOOL ;	//1-
   Me645 : BOOL ;	//1-
   Me646 : BOOL ;	//1-
   Me647 : BOOL ;	//1-
   Me648 : BOOL ;	//1-
   Me649 : BOOL ;	//1-
   Me650 : BOOL ;	//1-
   Me651 : BOOL ;	//1-
   Me652 : BOOL ;	//1-
   Me653 : BOOL ;	//1-
   Me654 : BOOL ;	//1-
   Me655 : BOOL ;	//1-
   Me656 : BOOL ;	//1-
   Me657 : BOOL ;	//1-
   Me658 : BOOL ;	//1-
   Me659 : BOOL ;	//1-
   Me660 : BOOL ;	//1-
   Me661 : BOOL ;	//1-
   Me662 : BOOL ;	//1-
   Me663 : BOOL ;	//1-
   Me664 : BOOL ;	//1-
   Me665 : BOOL ;	//1-
   Me666 : BOOL ;	//1-
   Me667 : BOOL ;	//1-
   Me668 : BOOL ;	//1-
   Me669 : BOOL ;	//1-
   Me670 : BOOL ;	//1-
   Me671 : BOOL ;	//1-
   Me672 : BOOL ;	//1-
   Me673 : BOOL ;	//1-
   Me674 : BOOL ;	//1-
   Me675 : BOOL ;	//1-
   Me676 : BOOL ;	//1-
   Me677 : BOOL ;	//1-
   Me678 : BOOL ;	//1-
   Me679 : BOOL ;	//1-
   Me680 : BOOL ;	//1-
   Me681 : BOOL ;	//1-
   Me682 : BOOL ;	//1-
   Me683 : BOOL ;	//1-
   Me684 : BOOL ;	//1-
   Me685 : BOOL ;	//1-
   Me686 : BOOL ;	//1-
   Me687 : BOOL ;	//1-
   Me688 : BOOL ;	//1-
   Me689 : BOOL ;	//1-
   Me690 : BOOL ;	//1-
   Me691 : BOOL ;	//1-
   Me692 : BOOL ;	//1-
   Me693 : BOOL ;	//1-
   Me694 : BOOL ;	//1-
   Me695 : BOOL ;	//1-
   Me696 : BOOL ;	//1-
   Me697 : BOOL ;	//1-
   Me698 : BOOL ;	//1-
   Me699 : BOOL ;	//1-
   Me700 : BOOL ;	//1-
   Me701 : BOOL ;	//1-
   Me702 : BOOL ;	//1-
   Me703 : BOOL ;	//1-
   Me704 : BOOL ;	//1-
   Me705 : BOOL ;	//1-
   Me706 : BOOL ;	//1-
   Me707 : BOOL ;	//1-
   Me708 : BOOL ;	//1-
   Me709 : BOOL ;	//1-
   Me710 : BOOL ;	//1-
   Me711 : BOOL ;	//1-
   Me712 : BOOL ;	//1-
   Me713 : BOOL ;	//1-
   Me714 : BOOL ;	//1-
   Me715 : BOOL ;	//1-
   Me716 : BOOL ;	//1-
   Me717 : BOOL ;	//1-
   Me718 : BOOL ;	//1-
   Me719 : BOOL ;	//1-
   Me720 : BOOL ;	//1-
   Me721 : BOOL ;	//1-
   Me722 : BOOL ;	//1-
   Me723 : BOOL ;	//1-
   Me724 : BOOL ;	//1-
   Me725 : BOOL ;	//1-
   Me726 : BOOL ;	//1-
   Me727 : BOOL ;	//1-
   Me728 : BOOL ;	//1-
   Me729 : BOOL ;	//1-
   Me730 : BOOL ;	//1-
   Me731 : BOOL ;	//1-
   Me732 : BOOL ;	//1-
   Me733 : BOOL ;	//1-
   Me734 : BOOL ;	//1-
   Me735 : BOOL ;	//1-
   Me736 : BOOL ;	//1-
   Me737 : BOOL ;	//1-
   Me738 : BOOL ;	//1-
   Me739 : BOOL ;	//1-
   Me740 : BOOL ;	//1-
   Me741 : BOOL ;	//1-
   Me742 : BOOL ;	//1-
   Me743 : BOOL ;	//1-
   Me744 : BOOL ;	//1-
   Me745 : BOOL ;	//1-
   Me746 : BOOL ;	//1-
   Me747 : BOOL ;	//1-
   Me748 : BOOL ;	//1-
   Me749 : BOOL ;	//1-
   Me750 : BOOL ;	//1-
   Me751 : BOOL ;	//1-
   Me752 : BOOL ;	//1-
   Me753 : BOOL ;	//1-
   Me754 : BOOL ;	//1-
   Me755 : BOOL ;	//1-
   Me756 : BOOL ;	//1-
   Me757 : BOOL ;	//1-
   Me758 : BOOL ;	//1-
   Me759 : BOOL ;	//1-
   Me760 : BOOL ;	//1-
   Me761 : BOOL ;	//1-
   Me762 : BOOL ;	//1-
   Me763 : BOOL ;	//1-
   Me764 : BOOL ;	//1-
   Me765 : BOOL ;	//1-
   Me766 : BOOL ;	//1-
   Me767 : BOOL ;	//1-
   Me768 : BOOL ;	//1-
   Me769 : BOOL ;	//1-
   Me770 : BOOL ;	//1-
   Me771 : BOOL ;	//1-
   Me772 : BOOL ;	//1-
   Me773 : BOOL ;	//1-
   Me774 : BOOL ;	//1-
   Me775 : BOOL ;	//1-
   Me776 : BOOL ;	//1-
   Me777 : BOOL ;	//1-
   Me778 : BOOL ;	//1-
   Me779 : BOOL ;	//1-
   Me780 : BOOL ;	//1-
   Me781 : BOOL ;	//1-
   Me782 : BOOL ;	//1-
   Me783 : BOOL ;	//1-
   Me784 : BOOL ;	//1-
   Me785 : BOOL ;	//1-
   Me786 : BOOL ;	//1-
   Me787 : BOOL ;	//1-
   Me788 : BOOL ;	//1-
   Me789 : BOOL ;	//1-
   Me790 : BOOL ;	//1-
   Me791 : BOOL ;	//1-
   Me792 : BOOL ;	//1-
   Me793 : BOOL ;	//1-
   Me794 : BOOL ;	//1-
   Me795 : BOOL ;	//1-
   Me796 : BOOL ;	//1-
   Me797 : BOOL ;	//1-
   Me798 : BOOL ;	//1-
   Me799 : BOOL ;	//1-
   Me800 : BOOL ;	//1-
   Me801 : BOOL ;	//1-
   Me802 : BOOL ;	//1-
   Me803 : BOOL ;	//1-
   Me804 : BOOL ;	//1-
   Me805 : BOOL ;	//1-
   Me806 : BOOL ;	//1-
   Me807 : BOOL ;	//1-
   Me808 : BOOL ;	//1-
   Me809 : BOOL ;	//1-
   Me810 : BOOL ;	//1-
   Me811 : BOOL ;	//1-
   Me812 : BOOL ;	//1-
   Me813 : BOOL ;	//1-
   Me814 : BOOL ;	//1-
   Me815 : BOOL ;	//1-
   Me816 : BOOL ;	//1-
   Me817 : BOOL ;	//1-
   Me818 : BOOL ;	//1-
   Me819 : BOOL ;	//1-
   Me820 : BOOL ;	//1-
   Me821 : BOOL ;	//1-
   Me822 : BOOL ;	//1-
   Me823 : BOOL ;	//1-
   Me824 : BOOL ;	//1-
   Me825 : BOOL ;	//1-
   Me826 : BOOL ;	//1-
   Me827 : BOOL ;	//1-
   Me828 : BOOL ;	//1-
   Me829 : BOOL ;	//1-
   Me830 : BOOL ;	//1-
   Me831 : BOOL ;	//1-
   Me832 : BOOL ;	//1-
   Me833 : BOOL ;	//1-
   Me834 : BOOL ;	//1-
   Me835 : BOOL ;	//1-
   Me836 : BOOL ;	//1-
   Me837 : BOOL ;	//1-
   Me838 : BOOL ;	//1-
   Me839 : BOOL ;	//1-
   Me840 : BOOL ;	//1-
   Me841 : BOOL ;	//1-
   Me842 : BOOL ;	//1-
   Me843 : BOOL ;	//1-
   Me844 : BOOL ;	//1-
   Me845 : BOOL ;	//1-
   Me846 : BOOL ;	//1-
   Me847 : BOOL ;	//1-
   Me848 : BOOL ;	//1-
   Me849 : BOOL ;	//1-
   Me850 : BOOL ;	//1-
   Me851 : BOOL ;	//1-
   Me852 : BOOL ;	//1-
   Me853 : BOOL ;	//1-
   Me854 : BOOL ;	//1-
   Me855 : BOOL ;	//1-
   Me856 : BOOL ;	//1-
   Me857 : BOOL ;	//1-
   Me858 : BOOL ;	//1-
   Me859 : BOOL ;	//1-
   Me860 : BOOL ;	//1-
   Me861 : BOOL ;	//1-
   Me862 : BOOL ;	//1-
   Me863 : BOOL ;	//1-
   Me864 : BOOL ;	//1-
   Me865 : BOOL ;	//1-
   Me866 : BOOL ;	//1-
   Me867 : BOOL ;	//1-
   Me868 : BOOL ;	//1-
   Me869 : BOOL ;	//1-
   Me870 : BOOL ;	//1-
   Me871 : BOOL ;	//1-
   Me872 : BOOL ;	//1-
   Me873 : BOOL ;	//1-
   Me874 : BOOL ;	//1-
   Me875 : BOOL ;	//1-
   Me876 : BOOL ;	//1-
   Me877 : BOOL ;	//1-
   Me878 : BOOL ;	//1-
   Me879 : BOOL ;	//1-
   Me880 : BOOL ;	//1-
   Me881 : BOOL ;	//1-
   Me882 : BOOL ;	//1-
   Me883 : BOOL ;	//1-
   Me884 : BOOL ;	//1-
   Me885 : BOOL ;	//1-
   Me886 : BOOL ;	//1-
   Me887 : BOOL ;	//1-
   Me888 : BOOL ;	//1-
   Me889 : BOOL ;	//1-
   Me890 : BOOL ;	//1-
   Me891 : BOOL ;	//1-
   Me892 : BOOL ;	//1-
   Me893 : BOOL ;	//1-
   Me894 : BOOL ;	//1-
   Me895 : BOOL ;	//1-
   Me896 : BOOL ;	//1-
   Me897 : BOOL ;	//1-
   Me898 : BOOL ;	//1-
   Me899 : BOOL ;	//1-
   Me900 : BOOL ;	//1-
   Me901 : BOOL ;	//1-
   Me902 : BOOL ;	//1-
   Me903 : BOOL ;	//1-
   Me904 : BOOL ;	//1-
   Me905 : BOOL ;	//1-
   Me906 : BOOL ;	//1-
   Me907 : BOOL ;	//1-
   Me908 : BOOL ;	//1-
   Me909 : BOOL ;	//1-
   Me910 : BOOL ;	//1-
   Me911 : BOOL ;	//1-
   Me912 : BOOL ;	//1-
   Me913 : BOOL ;	//1-
   Me914 : BOOL ;	//1-
   Me915 : BOOL ;	//1-
   Me916 : BOOL ;	//1-
   Me917 : BOOL ;	//1-
   Me918 : BOOL ;	//1-
   Me919 : BOOL ;	//1-
   Me920 : BOOL ;	//1-
   Me921 : BOOL ;	//1-
   Me922 : BOOL ;	//1-
   Me923 : BOOL ;	//1-
   Me924 : BOOL ;	//1-
   Me925 : BOOL ;	//1-
   Me926 : BOOL ;	//1-
   Me927 : BOOL ;	//1-
   Me928 : BOOL ;	//1-
   Me929 : BOOL ;	//1-
   Me930 : BOOL ;	//1-
   Me931 : BOOL ;	//1-
   Me932 : BOOL ;	//1-
   Me933 : BOOL ;	//1-
   Me934 : BOOL ;	//1-
   Me935 : BOOL ;	//1-
   Me936 : BOOL ;	//1-
   Me937 : BOOL ;	//1-
   Me938 : BOOL ;	//1-
   Me939 : BOOL ;	//1-
   Me940 : BOOL ;	//1-
   Me941 : BOOL ;	//1-
   Me942 : BOOL ;	//1-
   Me943 : BOOL ;	//1-
   Me944 : BOOL ;	//1-
   Me945 : BOOL ;	//1-
   Me946 : BOOL ;	//1-
   Me947 : BOOL ;	//1-
   Me948 : BOOL ;	//1-
   Me949 : BOOL ;	//1-
   Me950 : BOOL ;	//1-
   Me951 : BOOL ;	//1-
   Me952 : BOOL ;	//1-
   Me953 : BOOL ;	//1-
   Me954 : BOOL ;	//1-
   Me955 : BOOL ;	//1-
   Me956 : BOOL ;	//1-
   Me957 : BOOL ;	//1-
   Me958 : BOOL ;	//1-
   Me959 : BOOL ;	//1-
   Me960 : BOOL ;	//1-
   Me961 : BOOL ;	//1-
   Me962 : BOOL ;	//1-
   Me963 : BOOL ;	//1-
   Me964 : BOOL ;	//1-
   Me965 : BOOL ;	//1-
   Me966 : BOOL ;	//1-
   Me967 : BOOL ;	//1-
   Me968 : BOOL ;	//1-
   Me969 : BOOL ;	//1-
   Me970 : BOOL ;	//1-
   Me971 : BOOL ;	//1-
   Me972 : BOOL ;	//1-
   Me973 : BOOL ;	//1-
   Me974 : BOOL ;	//1-
   Me975 : BOOL ;	//1-
   Me976 : BOOL ;	//1-
   Me977 : BOOL ;	//1-
   Me978 : BOOL ;	//1-
   Me979 : BOOL ;	//1-
   Me980 : BOOL ;	//1-
   Me981 : BOOL ;	//1-
   Me982 : BOOL ;	//1-
   Me983 : BOOL ;	//1-
   Me984 : BOOL ;	//1-
   Me985 : BOOL ;	//1-
   Me986 : BOOL ;	//1-
   Me987 : BOOL ;	//1-
   Me988 : BOOL ;	//1-
   Me989 : BOOL ;	//1-
   Me990 : BOOL ;	//1-
   Me991 : BOOL ;	//1-
   Me992 : BOOL ;	//1-
   Me993 : BOOL ;	//1-
   Me994 : BOOL ;	//1-
   Me995 : BOOL ;	//1-
   Me996 : BOOL ;	//1-
   Me997 : BOOL ;	//1-
   Me998 : BOOL ;	//1-
   Me999 : BOOL ;	//1-
   Me1000 : BOOL ;	//1-
   Me1001 : BOOL ;	//1-
   Me1002 : BOOL ;	//1-
   Me1003 : BOOL ;	//1-
   Me1004 : BOOL ;	//1-
   Me1005 : BOOL ;	//1-
   Me1006 : BOOL ;	//1-
   Me1007 : BOOL ;	//1-
   Me1008 : BOOL ;	//1-
   Me1009 : BOOL ;	//1-
   Me1010 : BOOL ;	//1-
   Me1011 : BOOL ;	//1-
   Me1012 : BOOL ;	//1-
   Me1013 : BOOL ;	//1-
   Me1014 : BOOL ;	//1-
   Me1015 : BOOL ;	//1-
   Me1016 : BOOL ;	//1-
   Me1017 : BOOL ;	//1-
   Me1018 : BOOL ;	//1-
   Me1019 : BOOL ;	//1-
   Me1020 : BOOL ;	//1-
   Me1021 : BOOL ;	//1-
   Me1022 : BOOL ;	//1-
   Me1023 : BOOL ;	//1-
   Me1024 : BOOL ;	//1-
  END_STRUCT ;	
BEGIN
END_DATA_BLOCK

DATA_BLOCK "INST_DB_TOOLING_SYSTEM"	// DB 15
AUTHOR : A.Petz
VERSION : 0.0
"TOOLING SYSTEM???"
BEGIN
END_DATA_BLOCK

DATA_BLOCK "DB_COOLANT"	// DB 50
TITLE = Arbeitsdaten von FC_COOLANT
VERSION : 0.1
  STRUCT
   PSoll : INT ;	//stat:letzter gespeicherter KmSolldruck
   PSollAlt : INT ;	//stat:letzter gespeich.KmSolldruck (alt, für Änderungserfassung)
   PSollAA : INT ;	//stat:letzter gespeich.KmSolldruck, berechnet für AA
   P20AA : INT ;	//stat:Solldruck 20Bar, berechnet für AA
   P40AA : INT ;	//stat:Solldruck 40Bar, berechnet für AA
   fk : ARRAY  [0 .. 15 ] OF //stat:Flankenhilfsmerker
   BOOL ;
   hvFEin : BOOL ;	//stat:KmHauptventil Fehler:Einschaltüberwachung
   hvFUnt : BOOL ;	//stat:KmHauptventil Fehler:Unterbrechungsüberwachung
   kmdFEin : BOOL ;	//stat:KmSystem=Niederdruck Fehler:Einschaltüberwachung
   kmdFUnt : BOOL ;	//stat:KmSystem=Niederdruck Fehler:Unterbrechungsüberwachung
   FlFEin : BOOL ;	//stat:KmDurchfluss Fehler:Einschaltüberwachung
   FlFUnt : BOOL ;	//stat:KmDurchfluss Fehler:Unterbrechungsüberwachung
   x6 : BOOL ;
   x7 : BOOL ;
   x8 : BOOL ;
   x9 : BOOL ;
   x10 : BOOL ;
   x11 : BOOL ;
   x12 : BOOL ;
   x13 : BOOL ;
   x14 : BOOL ;
   x15 : BOOL ;
  END_STRUCT ;	
BEGIN
END_DATA_BLOCK

DATA_BLOCK "INS_MESSAGE_OUT"	// DB 100
AUTHOR : SPAC_slh
VERSION : 0.0
"MESSAGE_OUT"
BEGIN
END_DATA_BLOCK

DATA_BLOCK "DB_CK_OP"	// DB 101
VERSION : 0.1
  STRUCT
   T : ARRAY  [0 .. 31 ] OF UDT 1010;
  END_STRUCT ;	
BEGIN
END_DATA_BLOCK

DATA_BLOCK "DB_IN"	// DB 111
AUTHOR : APetz
VERSION : 0.1
  STRUCT
   EMX_MACHINE_ON : BOOL ;	//Maschine ist eingeschaltet (KEIN Not-Aus)
   EMX_WORKROOM_DOOR : BOOL ;	//Arbeitsraumtüre(n) der Werkzeugmaschine geschlossen und verriegelt
   EMX_ALARM_RESET : BOOL ;	//Meldung quittieren
   frei03 : BOOL ;
   EMX_COOLANT_BACKFLOW : BOOL ;	//Förderpumpe Sammelbehälter (Rückförderung aus Maschine)
   EMX_PNEUMATIC_PRESSURE : BOOL ;	//Systemdruck (pneumatik) vorhanden
   frei06 : BOOL ;
   frei07 : BOOL ;
   EMX_STROBE_COO_PRESSURE : BOOL ;	//Positiver Impuls zur Übernahme der benötigten Druckstufe
   frei11 : BOOL ;
   frei12 : BOOL ;
   frei13 : BOOL ;
   frei14 : BOOL ;
   frei15 : BOOL ;
   frei16 : BOOL ;
   frei17 : BOOL ;
   EMX_COOLANT1_M8 : BOOL ;	//Anforderung Kühlmittel_1 (M8 = AKZ)
   EMX_COOLANT2_M7 : BOOL ;	//Anforderung Kühlmittel_2 (M7 = IKZ)
   EMX_SPRAYGUN : BOOL ;	//Anforderung für Spülpistole
   EMX_FLUSH_LASERCOVER : BOOL ;	//Anforderung für die Spülung der Abdeckung Laser-Vermessung
   EMX_FLUSH_WORKPIECE1 : BOOL ;	//Anforderung für Dachspülung
   EMX_FLUSH_PALLET_CARRIER : BOOL ;	//Anforderung zum Abspülen der Auflageflächen der Palette am Palettenträger
   EMX_FLUSH_WORKROOMDOOR : BOOL ;	//Anforderung zur Reinigung der Arbeitsraumtüre
   QpxFlushSetUpStation : BOOL ;	//Anforderung von der Rüstplatzspülung
   frei30 : BOOL ;
   frei31 : BOOL ;
   frei32 : BOOL ;
   frei33 : BOOL ;
   frei34 : BOOL ;
   frei35 : BOOL ;
   frei36 : BOOL ;
   frei37 : BOOL ;
   EMX_COO_PRESSURE_BIT0 : BOOL ;	//Druckstufe BIT_0 = 1 (BCD-Code)
   EMX_COO_PRESSURE_BIT1 : BOOL ;	//Druckstufe BIT_1 = 2 (BCD-Code)
   EMX_COO_PRESSURE_BIT2 : BOOL ;	//Druckstufe BIT_2 = 4 (BCD-Code)
   EMX_COO_PRESSURE_BIT3 : BOOL ;	//Druckstufe BIT_3 = 8 (BCD-Code)
   EMX_COO_PRESSURE_BIT4 : BOOL ;	//Druckstufe BIT_4 = 10 (BCD-Code)
   EMX_COO_PRESSURE_BIT5 : BOOL ;	//Druckstufe BIT_5 = 20 (BCD-Code)
   EMX_COO_PRESSURE_BIT6 : BOOL ;	//Druckstufe BIT_6 = 40 (BCD-Code)
   EMX_COO_PRESSURE_BIT7 : BOOL ;	//Druckstufe BIT_7 = 80 (BCD-Code)
   frei50 : BOOL ;
   frei51 : BOOL ;
   frei52 : BOOL ;
   frei53 : BOOL ;
   frei54 : BOOL ;
   frei55 : BOOL ;
   frei56 : BOOL ;
   frei57 : BOOL ;
   EMW_PARAMETER_1 : WORD ;	//Konfiguration über Maschinenparameter_1
  END_STRUCT ;	
BEGIN
END_DATA_BLOCK

DATA_BLOCK "DB_OUT"	// DB 112
AUTHOR : APetz
VERSION : 0.1
  STRUCT
   AMX_ACK_COOLANT1_M8 : BOOL ;	//Quittiermeldung für Kühlmittel_1 (M8 = AKZ) ein (z.B. Pumpe läuft)
   AMX_ACK_COOLANT2_M7 : BOOL ;	//Quittiermeldung für Kühlmittel_2 (M7 = IKZ) ein (z.B. Pumpe läuft)
   AMX_MESSAGE_FLAG : BOOL ;	//Low-Signal, wenn an AW4 nur eine Warnung ansteht
   AMX_NO_EMERGENCY_STOP : BOOL ;	//FEHLER --> LOW-Signal löst ein Not-Aus der Werkzeugmaschine aus
   AMX_NO_SPINDLE_FEED_STP : BOOL ;	//FEHLER --> LOW_Pegel veranlasst Spindel- und Vorschub Halt
   AMX_NO_SPINDLE_FEED_STP0 : BOOL ;	//FEHLER --> LOW_Pegel veranlasst Spindel- und Vorschub Halt bei nächstem G0
   AMX_NO_DIAGNOSTIC_ALARM : BOOL ;	//FEHLER --> LOW-Signal, wenn Diagnoseeingang eines DESINA-Schalters nicht vorhan
   AMX_COO_MODE_AUTO : BOOL ;	//High-Signal, wenn die Kühlschmierstoffanlage in der Betriebsart AUTOMATIK ist
   AMX_CIRCUIT_OPEN_STOP : BOOL ;	//FEHLER --> LOW-Signal wenn Leistungsschalter ausgelöst - Maschine Stopp
   AMX_CIRCUIT_OPEN_MESSAGE : BOOL ;	//WARNUNG --> LOW-Signal wenn Leistungsschalter ausgelöst - Maschine läuft weiter
   AMX_COO_LEVEL_MAX : BOOL ;	//High-Signal, wenn der maximale Füllstand der KSA erreicht wird
   AMX_COO_LEVEL_MIN_MESSG : BOOL ;	//WARNUNG --> High-Signal, wenn ein Nachfüllen des Kühlmediums erforderlich ist
   AMX_COO_LEVEL_MIN_ALARM : BOOL ;	//FEHLER --> High-Signal, wenn minimaler Füllstand in KSA - Maschine Stopp
   AMX_PAPER_FILTER_END : BOOL ;	//FEHLER --> High-Signal, wenn Bandfilter Papier Ende - Maschine Stopp
   AMX_PAPER_FILTER_MESSG : BOOL ;	//WARNUNG --> High-Signal, Vorwarnung wenn Bandfilter Papier Minimum
   frei17 : BOOL ;
   frei20 : BOOL ;
   frei21 : BOOL ;
   frei22 : BOOL ;
   frei23 : BOOL ;
   frei24 : BOOL ;
   frei25 : BOOL ;
   frei26 : BOOL ;
   frei27 : BOOL ;
   frei30 : BOOL ;
   frei31 : BOOL ;
   frei32 : BOOL ;
   frei33 : BOOL ;
   frei34 : BOOL ;
   frei35 : BOOL ;
   frei36 : BOOL ;
   frei37 : BOOL ;
   AMW_MESSAGENUMBER : INT ;	//Meldungsnummer aus Sonderoption
   AMX_ACKCOO_PRESSURE_BIT0 : BOOL ;	//Rückmeldung Druckstufe BIT_0 = 1 (BCD-Code)
   AMX_ACKCOO_PRESSURE_BIT1 : BOOL ;	//Rückmeldung Druckstufe BIT_1 = 2 (BCD-Code)
   AMX_ACKCOO_PRESSURE_BIT2 : BOOL ;	//Rückmeldung Druckstufe BIT_2 = 4 (BCD-Code)
   AMX_ACKCOO_PRESSURE_BIT3 : BOOL ;	//Rückmeldung Druckstufe BIT_3 = 8 (BCD-Code)
   AMX_ACKCOO_PRESSURE_BIT4 : BOOL ;	//Rückmeldung Druckstufe BIT_4 = 10 (BCD-Code)
   AMX_ACKCOO_PRESSURE_BIT5 : BOOL ;	//Rückmeldung Druckstufe BIT_5 = 20 (BCD-Code)
   AMX_ACKCOO_PRESSURE_BIT6 : BOOL ;	//Rückmeldung Druckstufe BIT_6 = 40 (BCD-Code)
   AMX_ACKCOO_PRESSURE_BIT7 : BOOL ;	//Rückmeldung Druckstufe BIT_7 = 80 (BCD-Code)
   frei70 : BOOL ;
   frei71 : BOOL ;
   frei72 : BOOL ;
   frei73 : BOOL ;
   frei74 : BOOL ;
   frei75 : BOOL ;
   frei76 : BOOL ;
   frei77 : BOOL ;
  END_STRUCT ;	
BEGIN
END_DATA_BLOCK

ORGANIZATION_BLOCK "CYCL_EXC"	// OB 1
TITLE = "Main Program Sweep (Cycle)"
AUTHOR : APetz
VERSION : 0.1
VAR_TEMP
  OB1_EV_CLASS : BYTE ;	//Bits 0-3 = 1 (Coming event), Bits 4-7 = 1 (Event class 1)
  OB1_SCAN_1 : BYTE ;	//1 (Cold restart scan 1 of OB 1), 3 (Scan 2-n of OB 1)
  OB1_PRIORITY : BYTE ;	//Priority of OB Execution
  OB1_OB_NUMBR : BYTE ;	//1 (Organization block 1, OB1)
  OB1_RESERVED_1 : BYTE ;	//Reserved for system
  OB1_RESERVED_2 : BYTE ;	//Reserved for system
  OB1_PREV_CYCLE : INT ;	//Cycle time of previous OB1 scan (milliseconds)
  OB1_MIN_CYCLE : INT ;	//Minimum cycle time of OB1 (milliseconds)
  OB1_MAX_CYCLE : INT ;	//Maximum cycle time of OB1 (milliseconds)
  OB1_DATE_TIME : DATE_AND_TIME ;	//Date and time OB1 started
  TMP_BIT_PRUEF : BOOL ;	//Auswahl durch Konfiguration (MP)
  TMP_BIT_FEHLER_ND : BOOL ;	//Fehler im Niederdruck
  TMP_BIT_FEHLER_HD : BOOL ;	//Fehler im Hochdruck
  TMP_BYT_OPTION : BYTE ;	//Optionsauswahl
  TMP_BYT_ZEIT_AN_ND : BYTE ;	//Zeitparameter für Ansprechverhalten Niederdruck
  TMP_BYT_ZEIT_AB_ND : BYTE ;	//Zeitparameter für Abschaltverhalten Niederdruck
  TMP_BYT_ZEIT_AN_HD : BYTE ;	//Zeitparameter für Ansprechverhalten Hochdruck
  TMP_BYT_ZEIT_AB_HD : BYTE ;	//Zeitparameter für Abschaltverhalten Hochdruck
END_VAR
BEGIN
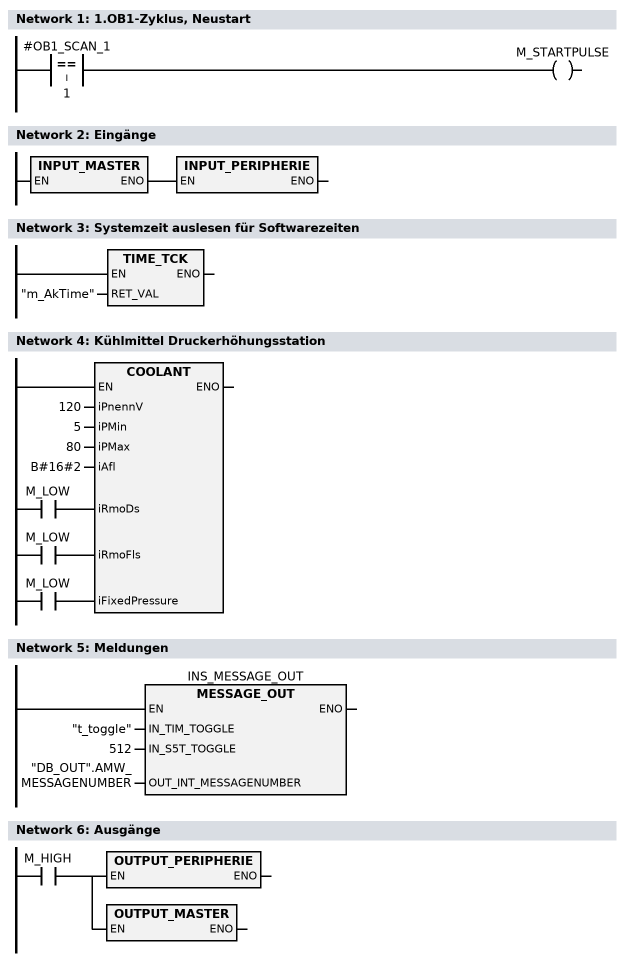
NETWORK
TITLE = 1.OB1-Zyklus, Neustart
//Eingänge von Mastersystem einlesen
//Eingänge von Peripherie lesen
      L     #OB1_SCAN_1;
      L     1;
      ==I;
      =     "M_STARTPULSE";
NETWORK
TITLE = Eingänge
//Eingänge von Mastersystem einlesen
//Eingänge von Peripherie lesen
      A(;
      CALL  "INPUT_MASTER";
      A     BR;
      );
      JNB   _001;
      CALL  "INPUT_PERIPHERIE";
_001: NOP   0;
NETWORK
TITLE = Systemzeit auslesen für Softwarezeiten
      CALL  "TIME_TCK" (
           RET_VAL                  := "m_AkTime");
      NOP   0;
NETWORK
TITLE = Kühlmittel Druckerhöhungsstation
      A     "M_LOW";
      =     L 26.0;
      BLD   103;
      A     "M_LOW";
      =     L 26.1;
      BLD   103;
      A     "M_LOW";
      =     L 26.2;
      BLD   103;
      CALL  "COOLANT" (
           iPnennV                  := 120,
           iPMin                    := 5,
           iPMax                    := 80,
           iAfl                     := B#16#2,
           iRmoDs                   := L 26.0,
           iRmoFls                  := L 26.1,
           iFixedPressure           := L 26.2);
      NOP   0;
NETWORK
TITLE = Meldungen
//Übergabe der Meldungen zum Master
//Wenn mehrere Meldungen anstehen, werden diese durchgetaktet
      CALL  "MESSAGE_OUT" , "INS_MESSAGE_OUT" (
           IN_TIM_TOGGLE            := "t_toggle",
           IN_S5T_TOGGLE            := 512,
           OUT_INT_MESSAGENUMBER    := "DB_OUT".AMW_MESSAGENUMBER);
      NOP   0;
NETWORK
TITLE = Ausgänge
//Ausgänge Peripherie schreiben
//Ausgänge an Mastersystem schreiben
      A     "M_HIGH";
      =     L 26.0;
      A     L 26.0;
      JNB   _002;
      CALL  "OUTPUT_PERIPHERIE";
_002: NOP   0;
      A     L 26.0;
      JNB   _003;
      CALL  "OUTPUT_MASTER";
_003: NOP   0;
END_ORGANIZATION_BLOCK

ORGANIZATION_BLOCK "I/O_FLT1"	// OB 82
TITLE = "I/O Point Fault"
VERSION : 0.1
VAR_TEMP
  OB82_EV_CLASS : BYTE ;	//16#39, Event class 3, Entering event state, Internal fault event
  OB82_FLT_ID : BYTE ;	//16#XX, Fault identifcation code
  OB82_PRIORITY : BYTE ;	//Priority of OB Execution
  OB82_OB_NUMBR : BYTE ;	//82 (Organization block 82, OB82)
  OB82_RESERVED_1 : BYTE ;	//Reserved for system
  OB82_IO_FLAG : BYTE ;	//Input (01010100), Output (01010101)
  OB82_MDL_ADDR : INT ;	//Base address of module with fault
  OB82_MDL_DEFECT : BOOL ;	//Module defective
  OB82_INT_FAULT : BOOL ;	//Internal fault
  OB82_EXT_FAULT : BOOL ;	//External fault
  OB82_PNT_INFO : BOOL ;	//Point information
  OB82_EXT_VOLTAGE : BOOL ;	//External voltage low
  OB82_FLD_CONNCTR : BOOL ;	//Field wiring connector missing
  OB82_NO_CONFIG : BOOL ;	//Module has no configuration data
  OB82_CONFIG_ERR : BOOL ;	//Module has configuration error
  OB82_MDL_TYPE : BYTE ;	//Type of module
  OB82_SUB_NDL_ERR : BOOL ;	//Sub-Module is missing or has error
  OB82_COMM_FAULT : BOOL ;	//Communication fault
  OB82_MDL_STOP : BOOL ;	//Module is stopped
  OB82_WTCH_DOG_FLT : BOOL ;	//Watch dog timer stopped module
  OB82_INT_PS_FLT : BOOL ;	//Internal power supply fault
  OB82_PRIM_BATT_FLT : BOOL ;	//Primary battery is in fault
  OB82_BCKUP_BATT_FLT : BOOL ;	//Backup battery is in fault
  OB82_RESERVED_2 : BOOL ;	//Reserved for system
  OB82_RACK_FLT : BOOL ;	//Rack fault, only for bus interface module
  OB82_PROC_FLT : BOOL ;	//Processor fault
  OB82_EPROM_FLT : BOOL ;	//EPROM fault
  OB82_RAM_FLT : BOOL ;	//RAM fault
  OB82_ADU_FLT : BOOL ;	//ADU fault
  OB82_FUSE_FLT : BOOL ;	//Fuse fault
  OB82_HW_INTR_FLT : BOOL ;	//Hardware interupt input in fault
  OB82_RESERVED_3 : BOOL ;	//Reserved for system
  OB82_DATE_TIME : DATE_AND_TIME ;	//Date and time OB82 started
END_VAR
BEGIN
NETWORK
TITLE =
END_ORGANIZATION_BLOCK

ORGANIZATION_BLOCK "OBNL_FLT"	// OB 85
TITLE = "Organization Block (OB) Not Loaded Fault"
VERSION : 0.1
VAR_TEMP
  OB85_EV_CLASS : BYTE ;	//16#35 Event class 3
  OB85_FLT_ID : BYTE ;	//16#XX, Fault identification code
  OB85_PRIORITY : BYTE ;	//Priority of OB Execution
  OB85_OB_NUMBR : BYTE ;	//85 (Organization block 85, OB85)
  OB85_RESERVED_1 : BYTE ;	//Reserved for system
  OB85_RESERVED_2 : BYTE ;	//Reserved for system
  OB85_RESERVED_3 : INT ;	//Reserved for system
  OB85_ERR_EV_CLASS : BYTE ;	//Class of event causing error
  OB85_ERR_EV_NUM : BYTE ;	//Number of event causing error
  OB85_OB_PRIOR : BYTE ;	//Priority of OB causing error
  OB85_OB_NUM : BYTE ;	//Number of OB causing error
  OB85_DATE_TIME : DATE_AND_TIME ;	//Date and time OB85 started
END_VAR
BEGIN
NETWORK
TITLE =
END_ORGANIZATION_BLOCK

ORGANIZATION_BLOCK "RACK_FLT"	// OB 86
TITLE = "Loss Of Rack Fault"
VERSION : 0.1
VAR_TEMP
  OB86_EV_CLASS : BYTE ;	//16#38/39 Event class 3
  OB86_FLT_ID : BYTE ;	//16#C1/C4/C5, Fault identifcation code
  OB86_PRIORITY : BYTE ;	//Priority of OB Execution
  OB86_OB_NUMBR : BYTE ;	//86 (Organization block 86, OB86)
  OB86_RESERVED_1 : BYTE ;	//Reserved for system
  OB86_RESERVED_2 : BYTE ;	//Reserved for system
  OB86_MDL_ADDR : INT ;	//Base address of IM module in rack with fault
  OB86_RACKS_FLTD : ARRAY  [0 .. 31 ] OF BOOL ;	//Racks in fault
  OB86_DATE_TIME : DATE_AND_TIME ;	//Date and time OB86 started
END_VAR
BEGIN
NETWORK
TITLE =
END_ORGANIZATION_BLOCK

ORGANIZATION_BLOCK "START"	// OB 100
TITLE = "Complete Restart"
VERSION : 0.1
VAR_TEMP
  OB100_EV_CLASS : BYTE ;	//16#13, Event class 1, Entering event state, Event logged in diagnostic buffer
  OB100_STRTUP : BYTE ;	//16#81/82/83/84 Method of startup
  OB100_PRIORITY : BYTE ;	//Priority of OB Execution
  OB100_OB_NUMBR : BYTE ;	//100 (Organization block 100, OB100)
  OB100_RESERVED_1 : BYTE ;	//Reserved for system
  OB100_RESERVED_2 : BYTE ;	//Reserved for system
  OB100_STOP : WORD ;	//Event that caused CPU to stop (16#4xxx)
  OB100_STRT_INFO : DWORD ;	//Information on how system started
  OB100_DATE_TIME : DATE_AND_TIME ;	//Date and time OB100 started
END_VAR
BEGIN
NETWORK
TITLE = Merker als Konstanten EINMALIG festlegen
//Bei KOP/FUP kann True oder False nicht als Konstante übergeben werden. Deshalb 
//definieren wir hier jeweils einen Merker, der immer true ist und einen Merker, 
//der immer false ist.
//Das Resetbit wird am Ende des OB1 sofort wieder zurückgesetzt, damit das 
//Resetbit nur für EINEN Zyklus ansteht.
      SET;
      R     "M_LOW";
      S     "M_HIGH";
      S     "m_inbetriebnahme";
END_ORGANIZATION_BLOCK

ORGANIZATION_BLOCK "PROG_ERR"	// OB 121
TITLE = "Programming Error"
VERSION : 0.1
VAR_TEMP
  OB121_EV_CLASS : BYTE ;	//16#25, Event class 2, Entering event state, Internal fault event
  OB121_SW_FLT : BYTE ;	//16#XX Software programming fault
  OB121_PRIORITY : BYTE ;	//Priority of OB Execution
  OB121_OB_NUMBR : BYTE ;	//121 (Organization block 121, OB121)
  OB121_BLK_TYPE : BYTE ;	//16#88/8A/8B/8C/8E Type of block fault occured in
  OB121_RESERVED_1 : BYTE ;	//Reserved for system
  OB121_FLT_REG : WORD ;	//16#XX Specific register that caused fault
  OB121_BLK_NUM : WORD ;	//Number of block that programming fault occured in
  OB121_PRG_ADDR : WORD ;	//Address in block where programming fault occured
  OB121_DATE_TIME : DATE_AND_TIME ;	//Date and time OB121 started
END_VAR
BEGIN
// (block stored without names or comments; labels and parameter names are numbered)
END_ORGANIZATION_BLOCK

ORGANIZATION_BLOCK "MOD_ERR"	// OB 122
TITLE = "Module Access Error"
VERSION : 0.1
VAR_TEMP
  OB122_EV_CLASS : BYTE ;	//16#29, Event class 2, Entering event state, Internal fault event
  OB122_SW_FLT : BYTE ;	//16#XX Software error code
  OB122_PRIORITY : BYTE ;	//Priority of OB Execution
  OB122_OB_NUMBR : BYTE ;	//122 (Organization block 122, OB122)
  OB122_BLK_TYPE : BYTE ;	//16#88/8C/8E Type of block fault occured in
  OB122_MEM_AREA : BYTE ;	//Memory area where access error occured
  OB122_MEM_ADDR : WORD ;	//Memory address where access error occured
  OB122_BLK_NUM : WORD ;	//Block number in which error occured
  OB122_PRG_ADDR : WORD ;	//Program address where error occured
  OB122_DATE_TIME : DATE_AND_TIME ;	//Date and time OB1 started
END_VAR
BEGIN
// (block stored without names or comments; labels and parameter names are numbered)
END_ORGANIZATION_BLOCK

